// TIA Portal V15.1 export
// export: Created 2024-06-21T08:41:15.862513Z, ExportSetting WithDefaults, DisplayName Totally Integrated Automation Portal, DisplayVersion V15.1 Update 5, DisplayName TIA Portal Openness, DisplayVersion V15.1 Update 5, DisplayName SINAMICS Startdrive Advanced, DisplayVersion V15.1, DisplayName G130, G150, S120, S150, SINAMICS MV, S210, DisplayVersion V15.1, DisplayName G110M, G120, G120C, G120D, G120P, DisplayVersion V15.1, DisplayName STEP 7 Professional, DisplayVersion V15.1 Update 5, DisplayName STEP 7 Safety, DisplayVersion V15.1, DisplayName WinCC Professional, DisplayVersion V15.1 Update 5, DisplayName SIMATIC Visualization Architect, DisplayVersion V15.1
FUNCTION_BLOCK "LGBHoist2Pos2S-C"   // FB6646, FBD
TITLE = LGBHoist2Pos2S-C
{ S7_Optimized_Access := 'TRUE' }
AUTHOR : VCC
FAMILY : Transpor
VERSION : 0.1
// =============================================================================
// This module is used in applications when a Hoist with 2 Positions and two Speeds controlled
// by contactors is needed.
// =============================================================================
// stored: AutoNumber false, IsIECCheckEnabled false, IsRetainMemResEnabled false, MemoryReserve 100, SetENOAutomatically False, UDAEnableTagReadback false
   VAR_INPUT
      I_OverTravelSet { ExternalAccessible := 'False'; ExternalVisible := 'False'; ExternalWritable := 'False'} : Bool;   // Overtravel Switch Set
      I_StopDetSet { ExternalAccessible := 'False'; ExternalVisible := 'False'; ExternalWritable := 'False'} : Bool;   // Stop Detection Set
      I_LowSpeedDetSet { ExternalAccessible := 'False'; ExternalVisible := 'False'; ExternalWritable := 'False'} : Bool;   // Lowspeed Detection Set
      I_LowSpeedDetSetCtrl { ExternalAccessible := 'False'; ExternalVisible := 'False'; ExternalWritable := 'False'} : Bool;   // Lowspeed Detection Set
      I_LowSpeedDetRes { ExternalAccessible := 'False'; ExternalVisible := 'False'; ExternalWritable := 'False'} : Bool;   // Lowspeed Detector Reset
      I_LowSpeedDetResCtrl { ExternalAccessible := 'False'; ExternalVisible := 'False'; ExternalWritable := 'False'} : Bool;   // Lowspeed Detector Reset
      I_StopDetRes { ExternalAccessible := 'False'; ExternalVisible := 'False'; ExternalWritable := 'False'} : Bool;   // Stop Detection Reset
      I_OverTravelRes { ExternalAccessible := 'False'; ExternalVisible := 'False'; ExternalWritable := 'False'} : Bool;   // Overtravel Switch Reset
      I_BypassOvertravelSet { ExternalAccessible := 'False'; ExternalVisible := 'False'; ExternalWritable := 'False'} : Bool;   // Bypass overtravel Set
      I_BypassOvertravelReset { ExternalAccessible := 'False'; ExternalVisible := 'False'; ExternalWritable := 'False'} : Bool;   // Bypass overtravel Reset
      I_BrakeReleased { ExternalAccessible := 'False'; ExternalVisible := 'False'; ExternalWritable := 'False'} : Bool;   // Feedback from brake contactor
      I_SetBegin { ExternalAccessible := 'False'; ExternalVisible := 'False'; ExternalWritable := 'False'} : Bool;   // Condition to start movement Set
      I_ResBegin { ExternalAccessible := 'False'; ExternalVisible := 'False'; ExternalWritable := 'False'} : Bool;   // Condition to start movement Reset
      I_InterlockSetOk { ExternalAccessible := 'False'; ExternalVisible := 'False'; ExternalWritable := 'False'} : Bool;   // Interlock Set Ok
      I_InterlockResetOk { ExternalAccessible := 'False'; ExternalVisible := 'False'; ExternalWritable := 'False'} : Bool;   // Interlock Reset Ok
      I_MotorProtection { ExternalAccessible := 'False'; ExternalVisible := 'False'; ExternalWritable := 'False'} : Bool;   // Motor protection
      I_SafetySwitch { ExternalAccessible := 'False'; ExternalVisible := 'False'; ExternalWritable := 'False'} : Bool;   // Safety Switch
      I_PBSet { ExternalAccessible := 'False'; ExternalVisible := 'False'; ExternalWritable := 'False'} : Bool;   // Push button for manual movememt (on local panel) Set
      I_PBReset { ExternalAccessible := 'False'; ExternalVisible := 'False'; ExternalWritable := 'False'} : Bool;   // Push button for manual movememt (on local panel) Reset
      I_SafetyOk { ExternalAccessible := 'False'; ExternalVisible := 'False'; ExternalWritable := 'False'} : Bool;   // Safety Ok
      I_MotionStopOk { ExternalAccessible := 'False'; ExternalVisible := 'False'; ExternalWritable := 'False'} : Bool;   // Safety Ok / The motion stop is Ok
   END_VAR
   VAR_OUTPUT
      O_SetContactor { ExternalAccessible := 'False'; ExternalVisible := 'False'; ExternalWritable := 'False'} : Bool;   // Activate set contactor / Activate Set Contactor
      O_ResetContactor { ExternalAccessible := 'False'; ExternalVisible := 'False'; ExternalWritable := 'False'} : Bool;   // Activate Reset contactor / Activate Reset Contactor
      O_HSpdContactor { ExternalAccessible := 'False'; ExternalVisible := 'False'; ExternalWritable := 'False'} : Bool;   // Activate High Speed contactor / Activate High Speed Contactor
      O_LSpdContactor { ExternalAccessible := 'False'; ExternalVisible := 'False'; ExternalWritable := 'False'} : Bool;   // Activate low speed contactor / Activate Low Speed Contactor
      O_ReleaseBrake { ExternalAccessible := 'False'; ExternalVisible := 'False'; ExternalWritable := 'False'} : Bool;   // Release the brake of the Motor
      O_ContBypassOvertravelSet { ExternalAccessible := 'False'; ExternalVisible := 'False'; ExternalWritable := 'False'} : Bool;   // Contactor Bypass overtravel Set
      O_ContBypassOvertravelRes { ExternalAccessible := 'False'; ExternalVisible := 'False'; ExternalWritable := 'False'} : Bool;   // Contactor Bypass overtravel Reset
      O_Active { ExternalAccessible := 'False'; ExternalVisible := 'False'; ExternalWritable := 'False'} : Bool;   // Hoist is active
      O_SetFinished { ExternalAccessible := 'False'; ExternalVisible := 'False'; ExternalWritable := 'False'} : Bool;   // Set Position finished
      O_ResFinished { ExternalAccessible := 'False'; ExternalVisible := 'False'; ExternalWritable := 'False'} : Bool;   // Reset Position finished
      O_InSetPos { ExternalAccessible := 'False'; ExternalVisible := 'False'; ExternalWritable := 'False'} : Bool;   // In set Position
      O_InResPos { ExternalAccessible := 'False'; ExternalVisible := 'False'; ExternalWritable := 'False'} : Bool;   // In Reset Position
      O_LEDSet { ExternalAccessible := 'False'; ExternalVisible := 'False'; ExternalWritable := 'False'} : Bool;   // Ledindication / Led indication for Set
      O_LEDRes { ExternalAccessible := 'False'; ExternalVisible := 'False'; ExternalWritable := 'False'} : Bool;   // Ledindication / Led indication for Reset
      O_AlarmABCondition { ExternalAccessible := 'False'; ExternalVisible := 'False'; ExternalWritable := 'False'} : Bool;   // Alarm AB Condition
      O_AlarmA { ExternalAccessible := 'False'; ExternalVisible := 'False'; ExternalWritable := 'False'} : Bool;   // Summation Alarm A
      O_AlarmB { ExternalAccessible := 'False'; ExternalVisible := 'False'; ExternalWritable := 'False'} : Bool;   // Summation Alarm B
      O_AlarmC { ExternalAccessible := 'False'; ExternalVisible := 'False'; ExternalWritable := 'False'} : Bool;   // Summation Alarm C
      O_AlarmD { ExternalAccessible := 'False'; ExternalVisible := 'False'; ExternalWritable := 'False'} : Bool;   // Summation Alarm D
      O_ActualSpeed { ExternalAccessible := 'False'; ExternalVisible := 'False'; ExternalWritable := 'False'} : Real;   // Actual speed value motor
      H_AlarmDWord { ExternalAccessible := 'False'; ExternalVisible := 'False'; ExternalWritable := 'False'} : DWord;   // HMI Alarm Word
   END_VAR
   VAR_IN_OUT
      C_TimeCheckSpeedOK { ExternalAccessible := 'False'; ExternalVisible := 'False'; ExternalWritable := 'False'} : DInt := 2000;   // Time check speed OK
      IO_Modes : "Modes";   // Modes
      H_HMI : "H_HMI";   // Animation
      "H_GBHoist2Pos2S-C" : "H_GBHoist2Pos2S-C";   // Animation
      C_Config : "Hoist2Pos2S-C-Config";   // Config
   END_VAR
   VAR
      _Motor { ExternalAccessible := 'False'; ExternalVisible := 'False'; ExternalWritable := 'False'} : "LGBMotor2W2S-C";
      H_FncSelInHMI { ExternalAccessible := 'False'; ExternalVisible := 'False'; ExternalWritable := 'False'} : Bool;
      AlarmABCondition { ExternalAccessible := 'False'; ExternalVisible := 'False'; ExternalWritable := 'False'} : Bool;   // Alarm AB Condition
      AA_MotorProtection { ExternalAccessible := 'False'; ExternalVisible := 'False'; ExternalWritable := 'False'} : Bool;   // Motorprotection Tripped
      AA_SafetySwitch { ExternalAccessible := 'False'; ExternalVisible := 'False'; ExternalWritable := 'False'} : Bool;   // Safety Switch Not Ok
      AB_OverTravelSet { ExternalAccessible := 'False'; ExternalVisible := 'False'; ExternalWritable := 'False'} : Bool;   // Overtravel Set
      AB_OverTravelRes { ExternalAccessible := 'False'; ExternalVisible := 'False'; ExternalWritable := 'False'} : Bool;   // Overtravel Reset
      AB_LSpDetSet { ExternalAccessible := 'False'; ExternalVisible := 'False'; ExternalWritable := 'False'} : Bool;   // Low Speed Detector Set Missing
      AB_LSpDetSetCtrl { ExternalAccessible := 'False'; ExternalVisible := 'False'; ExternalWritable := 'False'} : Bool;   // Low Speed Detector Ctrl Set Missing
      AB_LSpDetRes { ExternalAccessible := 'False'; ExternalVisible := 'False'; ExternalWritable := 'False'} : Bool;   // Low Speed Detector Reset Missing
      AB_LSpDetResCtrl { ExternalAccessible := 'False'; ExternalVisible := 'False'; ExternalWritable := 'False'} : Bool;   // Low Speed Detector Ctrl Reset Missing
      AB_BrakeFbk { ExternalAccessible := 'False'; ExternalVisible := 'False'; ExternalWritable := 'False'} : Bool;   // Safety Switch Not Ok / Brake feedback Nok / Säkerhetsbrytare Ej Ok
      AC_OvtSetAlm { ExternalAccessible := 'False'; ExternalVisible := 'False'; ExternalWritable := 'False'} : Bool;   // Timeout Set
      AC_OvtResAlm { ExternalAccessible := 'False'; ExternalVisible := 'False'; ExternalWritable := 'False'} : Bool;   // Timeout Reset
      AC_OvertravelSetBypassAlm { ExternalAccessible := 'False'; ExternalVisible := 'False'; ExternalWritable := 'False'} : Bool;   // Overtravel Set Bypass
      AC_OvertravelResBypassAlm { ExternalAccessible := 'False'; ExternalVisible := 'False'; ExternalWritable := 'False'} : Bool;   // Overtravel Reset Bypass
      AD_IntlkSet { ExternalAccessible := 'False'; ExternalVisible := 'False'; ExternalWritable := 'False'} : Bool;   // Interlock Not Ok
      AD_IntlkRes { ExternalAccessible := 'False'; ExternalVisible := 'False'; ExternalWritable := 'False'} : Bool;   // Interlock Not Ok
      AC_LiftNoPos { ExternalAccessible := 'False'; ExternalVisible := 'False'; ExternalWritable := 'False'} : Bool;   // Lifter Not in position
      AD_MotionStop { ExternalAccessible := 'False'; ExternalVisible := 'False'; ExternalWritable := 'False'} : Bool;   // Motion Stop
      SafetyOk { ExternalAccessible := 'False'; ExternalVisible := 'False'; ExternalWritable := 'False'} : Bool;   // Safety Ok
      AlarmA { ExternalAccessible := 'False'; ExternalVisible := 'False'; ExternalWritable := 'False'} : Bool;   // Alarm A
      AlarmB { ExternalAccessible := 'False'; ExternalVisible := 'False'; ExternalWritable := 'False'} : Bool;   // Alarm B
      AlarmC { ExternalAccessible := 'False'; ExternalVisible := 'False'; ExternalWritable := 'False'} : Bool;   // Alarm C
      AlarmD { ExternalAccessible := 'False'; ExternalVisible := 'False'; ExternalWritable := 'False'} : Bool;   // Alarm D
      LSpdContactor { ExternalAccessible := 'False'; ExternalVisible := 'False'; ExternalWritable := 'False'} : Bool;   // Contactor low speed / Activate Low Speed Contactor
      HSpdContactor { ExternalAccessible := 'False'; ExternalVisible := 'False'; ExternalWritable := 'False'} : Bool;   // Contactor High Speed / Activate High Speed Contactor
      SetContactor { ExternalAccessible := 'False'; ExternalVisible := 'False'; ExternalWritable := 'False'} : Bool;   // Activate Set Contactor
      ResetContactor { ExternalAccessible := 'False'; ExternalVisible := 'False'; ExternalWritable := 'False'} : Bool;   // Activate Reset Contactor
      ReleaseBrake { ExternalAccessible := 'False'; ExternalVisible := 'False'; ExternalWritable := 'False'} : Bool;   // Activate Reset contactor / Release Brake
      MotorLoopActive { ExternalAccessible := 'False'; ExternalVisible := 'False'; ExternalWritable := 'False'} : Bool;   // Motor Loop Active
      MotorCmdLSpdSet { ExternalAccessible := 'False'; ExternalVisible := 'False'; ExternalWritable := 'False'} : Bool;   // Command to Motorloop low Speed Set
      MotorCmdLSpdRes { ExternalAccessible := 'False'; ExternalVisible := 'False'; ExternalWritable := 'False'} : Bool;   // Command to Motorloop low speed Reset
      MotorCmdHSpdSet { ExternalAccessible := 'False'; ExternalVisible := 'False'; ExternalWritable := 'False'} : Bool;   // Command to Motorloop high Speed Set
      MotorCmdHSpdRes { ExternalAccessible := 'False'; ExternalVisible := 'False'; ExternalWritable := 'False'} : Bool;   // Command to Motorloop high speed Reset
      MotorReqLSpdSet { ExternalAccessible := 'False'; ExternalVisible := 'False'; ExternalWritable := 'False'} : Bool;   // Request low Speed Set
      MotorReqLSpdRes { ExternalAccessible := 'False'; ExternalVisible := 'False'; ExternalWritable := 'False'} : Bool;   // Request low speed Reset
      MotorReqHSpdSet { ExternalAccessible := 'False'; ExternalVisible := 'False'; ExternalWritable := 'False'} : Bool;   // Request highSpeed Set
      MotorReqHSpdRes { ExternalAccessible := 'False'; ExternalVisible := 'False'; ExternalWritable := 'False'} : Bool;   // Request high speed Reset
      ManHighSpdSel { ExternalAccessible := 'False'; ExternalVisible := 'False'; ExternalWritable := 'False'} : Bool;   // Low speed selected in manual
      HSpdMem { ExternalAccessible := 'False'; ExternalVisible := 'False'; ExternalWritable := 'False'} : Bool;   // High speed memory flag
      BlockHSpeed { ExternalAccessible := 'False'; ExternalVisible := 'False'; ExternalWritable := 'False'} : Bool;   // AND of ALL detections
      AlarmABAct { ExternalAccessible := 'False'; ExternalVisible := 'False'; ExternalWritable := 'False'} : Bool;   // Alarm A or B is active
      OverTravelSetAlmCond { ExternalAccessible := 'False'; ExternalVisible := 'False'; ExternalWritable := 'False'} : Bool;   // Alarm AB Condition
      OverTravelResAlmCond { ExternalAccessible := 'False'; ExternalVisible := 'False'; ExternalWritable := 'False'} : Bool;   // Alarm AB Condition
      MotorLoopAlmCond { ExternalAccessible := 'False'; ExternalVisible := 'False'; ExternalWritable := 'False'} : Bool;   // Alarm AB Condition
      CmdSet { ExternalAccessible := 'False'; ExternalVisible := 'False'; ExternalWritable := 'False'} : Bool;   // Activate Set (up) command
      CmdRes { ExternalAccessible := 'False'; ExternalVisible := 'False'; ExternalWritable := 'False'} : Bool;   // Activate Reset (down) command
      InSetPos { ExternalAccessible := 'False'; ExternalVisible := 'False'; ExternalWritable := 'False'} : Bool;   // In set Position
      InResPos { ExternalAccessible := 'False'; ExternalVisible := 'False'; ExternalWritable := 'False'} : Bool;   // In Reset Position
      TimeOutNotDownCmd { ExternalAccessible := 'False'; ExternalVisible := 'False'; ExternalWritable := 'False'} : Bool;   // Timer result
      TimeOutNotUpCmd { ExternalAccessible := 'False'; ExternalVisible := 'False'; ExternalWritable := 'False'} : Bool;   // Timer result
      _TimerNoDownCmd { ExternalAccessible := 'False'; ExternalVisible := 'False'; ExternalWritable := 'False'} : "LTimer";   // FB
      _TimerNoUpCmd { ExternalAccessible := 'False'; ExternalVisible := 'False'; ExternalWritable := 'False'} : "LTimer";   // FB
      _TimerNoPos { ExternalAccessible := 'False'; ExternalVisible := 'False'; ExternalWritable := 'False'} : "LTimer";
      _BypassOvertravelSet { ExternalAccessible := 'False'; ExternalVisible := 'False'; ExternalWritable := 'False'} : "L1AlarmMultiIn";   // FB
      _BypassOvertravelReset { ExternalAccessible := 'False'; ExternalVisible := 'False'; ExternalWritable := 'False'} : "L1AlarmMultiIn";   // FB
      _OverTravelSet { ExternalAccessible := 'False'; ExternalVisible := 'False'; ExternalWritable := 'False'} : "L1AlarmMultiIn";
      _OverTravelRes { ExternalAccessible := 'False'; ExternalVisible := 'False'; ExternalWritable := 'False'} : "L1AlarmMultiIn";
      _OvtSetAlmTimer { ExternalAccessible := 'False'; ExternalVisible := 'False'; ExternalWritable := 'False'} : "LTimer";   // FB
      _OvtResAlmTimer { ExternalAccessible := 'False'; ExternalVisible := 'False'; ExternalWritable := 'False'} : "LTimer";   // FB
      Edge { ExternalAccessible := 'False'; ExternalVisible := 'False'; ExternalWritable := 'False'} : Array[1..8] of Bool;   // Edge
   END_VAR
   VAR_TEMP
      NotUsedH_HMI : "H_HMI";   // Temp
      H_HMIMotor : "H_HMI";   // Temp
      HMICMD : "ConvHMICMD";   // Temp
   END_VAR
   VAR_TEMP   // added for the SCL form of the ladder/FBD networks
      _w1 : Bool;
   END_VAR
BEGIN

REGION Network 1: **** 1 - Inputs **** HMI Commands
   // HMI Commands
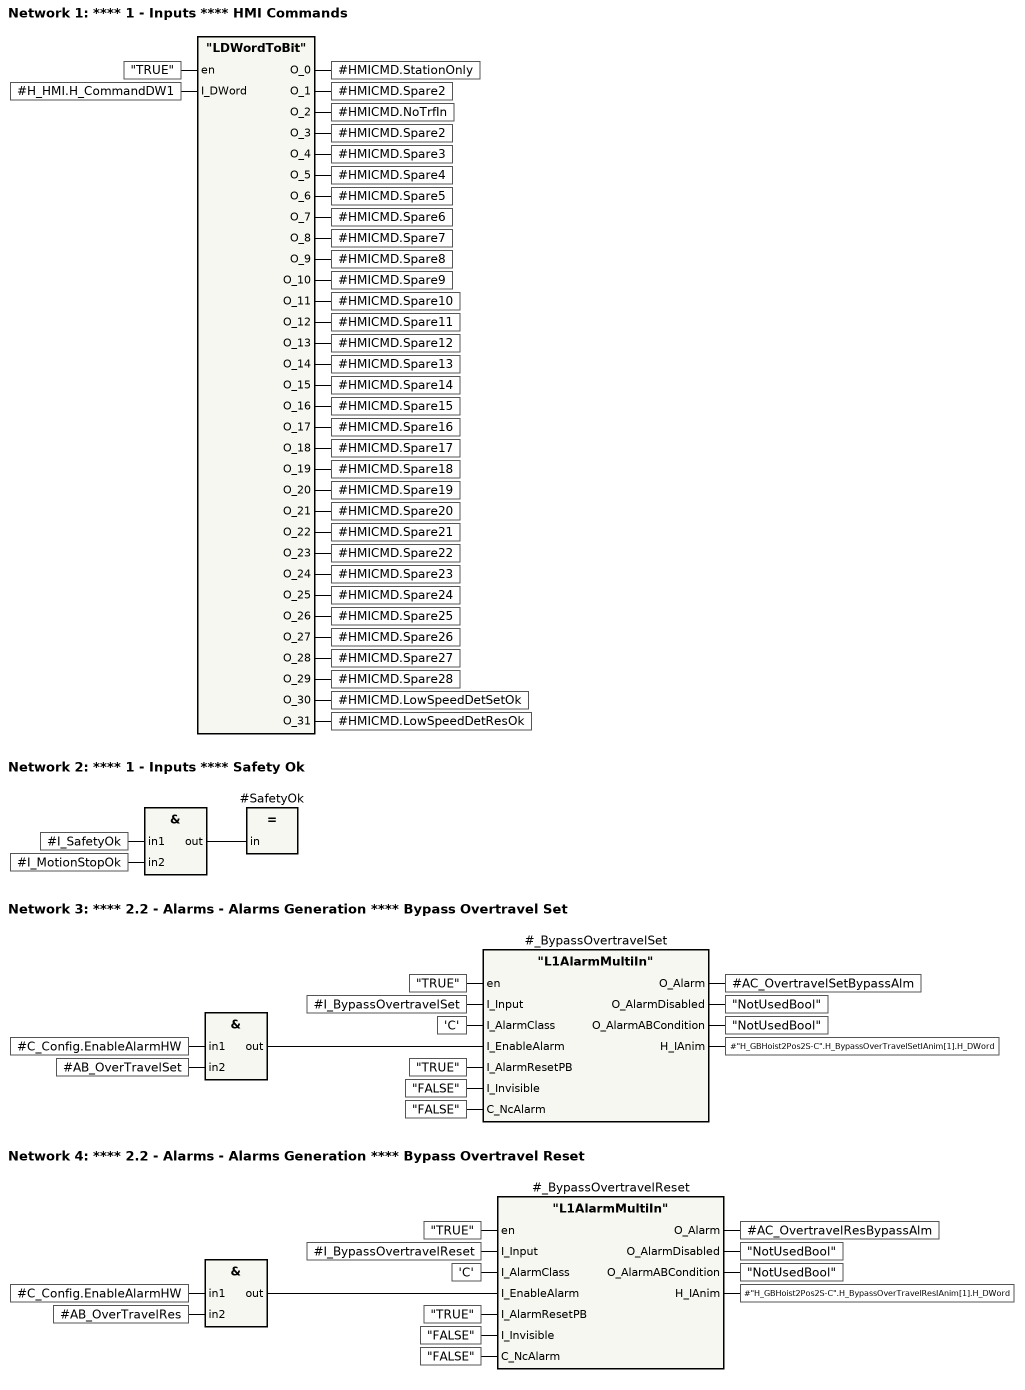
   IF "TRUE" THEN
       "LDWordToBit"(I_DWord := #H_HMI.H_CommandDW1,
                     O_0 => #HMICMD.StationOnly,
                     O_1 => #HMICMD.Spare2,
                     O_2 => #HMICMD.NoTrfIn,
                     O_3 => #HMICMD.Spare2,
                     O_4 => #HMICMD.Spare3,
                     O_5 => #HMICMD.Spare4,
                     O_6 => #HMICMD.Spare5,
                     O_7 => #HMICMD.Spare6,
                     O_8 => #HMICMD.Spare7,
                     O_9 => #HMICMD.Spare8,
                     O_10 => #HMICMD.Spare9,
                     O_11 => #HMICMD.Spare10,
                     O_12 => #HMICMD.Spare11,
                     O_13 => #HMICMD.Spare12,
                     O_14 => #HMICMD.Spare13,
                     O_15 => #HMICMD.Spare14,
                     O_16 => #HMICMD.Spare15,
                     O_17 => #HMICMD.Spare16,
                     O_18 => #HMICMD.Spare17,
                     O_19 => #HMICMD.Spare18,
                     O_20 => #HMICMD.Spare19,
                     O_21 => #HMICMD.Spare20,
                     O_22 => #HMICMD.Spare21,
                     O_23 => #HMICMD.Spare22,
                     O_24 => #HMICMD.Spare23,
                     O_25 => #HMICMD.Spare24,
                     O_26 => #HMICMD.Spare25,
                     O_27 => #HMICMD.Spare26,
                     O_28 => #HMICMD.Spare27,
                     O_29 => #HMICMD.Spare28,
                     O_30 => #HMICMD.LowSpeedDetSetOk,
                     O_31 => #HMICMD.LowSpeedDetResOk);
   END_IF;
END_REGION

REGION Network 2: **** 1 - Inputs **** Safety Ok
   #SafetyOk := #I_SafetyOk AND #I_MotionStopOk;
END_REGION

REGION Network 3: **** 2.2 - Alarms - Alarms Generation **** Bypass Overtravel Set
   // Alarm Bypass Overtravel Set
   IF "TRUE" THEN
       #_BypassOvertravelSet(I_Input := #I_BypassOvertravelSet,   // "L1AlarmMultiIn"
                             I_AlarmClass := 'C',
                             I_EnableAlarm := #C_Config.EnableAlarmHW AND #AB_OverTravelSet,
                             I_AlarmResetPB := "TRUE",
                             I_Invisible := "FALSE",
                             C_NcAlarm := "FALSE",
                             O_Alarm => #AC_OvertravelSetBypassAlm,
                             O_AlarmDisabled => "NotUsedBool",
                             O_AlarmABCondition => "NotUsedBool",
                             H_IAnim => #"H_GBHoist2Pos2S-C".H_BypassOverTravelSetIAnim[1].H_DWord);
   END_IF;
END_REGION

REGION Network 4: **** 2.2 - Alarms - Alarms Generation **** Bypass Overtravel Reset
   // Alarm Bypass Overtravel Reset
   IF "TRUE" THEN
       #_BypassOvertravelReset(I_Input := #I_BypassOvertravelReset,   // "L1AlarmMultiIn"
                               I_AlarmClass := 'C',
                               I_EnableAlarm := #C_Config.EnableAlarmHW AND #AB_OverTravelRes,
                               I_AlarmResetPB := "TRUE",
                               I_Invisible := "FALSE",
                               C_NcAlarm := "FALSE",
                               O_Alarm => #AC_OvertravelResBypassAlm,
                               O_AlarmDisabled => "NotUsedBool",
                               O_AlarmABCondition => "NotUsedBool",
                               H_IAnim => #"H_GBHoist2Pos2S-C".H_BypassOverTravelResIAnim[1].H_DWord);
   END_IF;
END_REGION

REGION Network 5: **** 2.2 - Alarms - Alarms Generation **** Over Travel Set Alarm
   // Over Travel Set Alarm
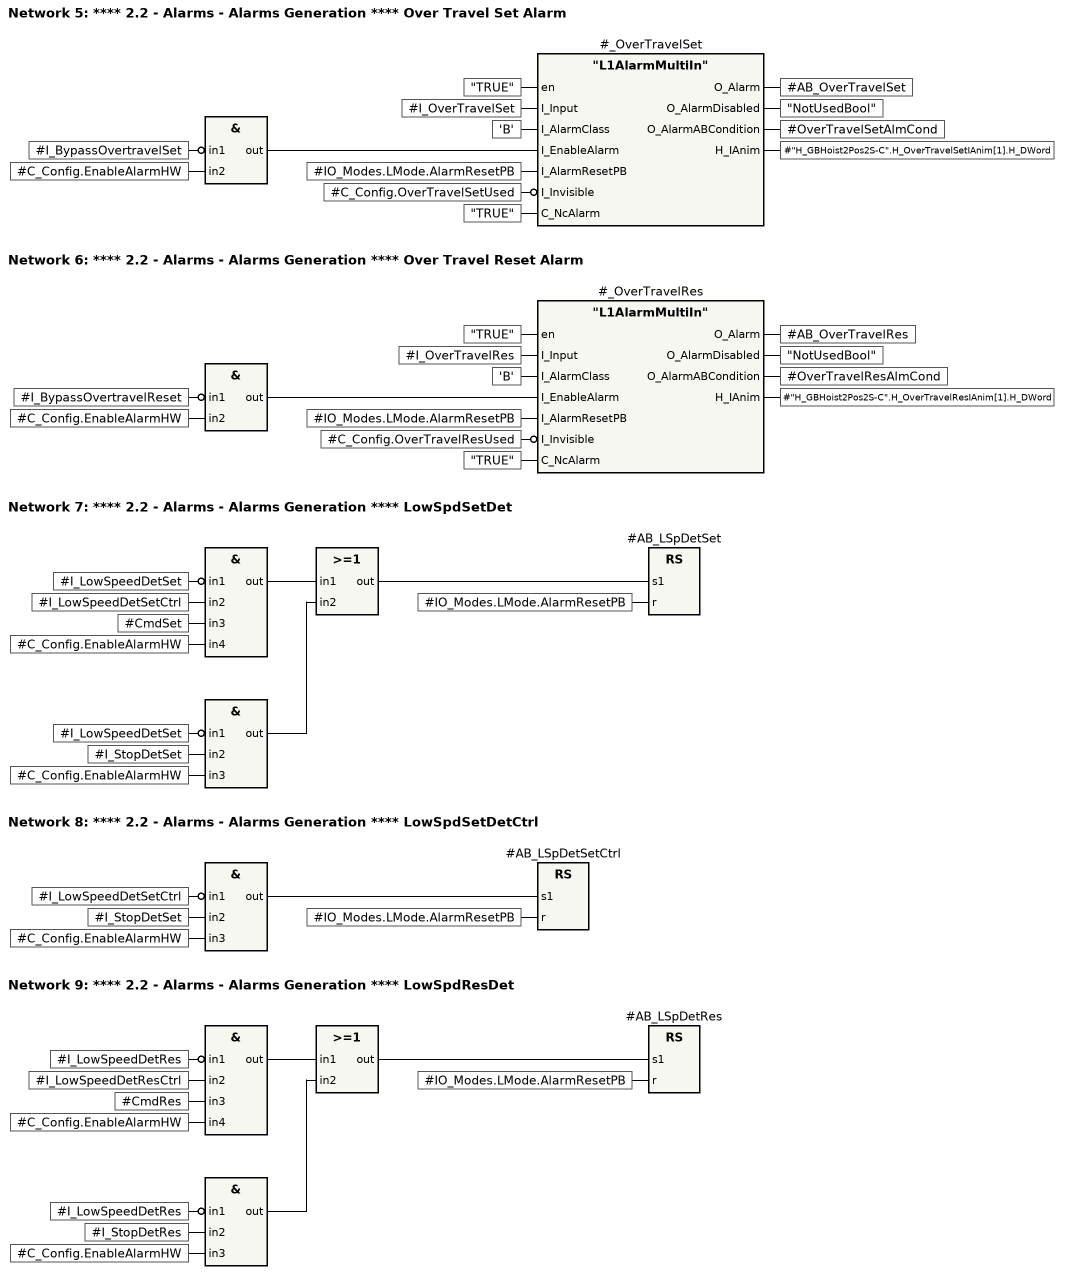
   IF "TRUE" THEN
       #_OverTravelSet(I_Input := #I_OverTravelSet,   // "L1AlarmMultiIn"
                       I_AlarmClass := 'B',
                       I_EnableAlarm := NOT #I_BypassOvertravelSet AND #C_Config.EnableAlarmHW,
                       I_AlarmResetPB := #IO_Modes.LMode.AlarmResetPB,
                       I_Invisible := NOT #C_Config.OverTravelSetUsed,
                       C_NcAlarm := "TRUE",
                       O_Alarm => #AB_OverTravelSet,
                       O_AlarmDisabled => "NotUsedBool",
                       O_AlarmABCondition => #OverTravelSetAlmCond,
                       H_IAnim => #"H_GBHoist2Pos2S-C".H_OverTravelSetIAnim[1].H_DWord);
   END_IF;
END_REGION

REGION Network 6: **** 2.2 - Alarms - Alarms Generation **** Over Travel Reset Alarm
   // Over Travel Reset Alarm
   IF "TRUE" THEN
       #_OverTravelRes(I_Input := #I_OverTravelRes,   // "L1AlarmMultiIn"
                       I_AlarmClass := 'B',
                       I_EnableAlarm := NOT #I_BypassOvertravelReset AND #C_Config.EnableAlarmHW,
                       I_AlarmResetPB := #IO_Modes.LMode.AlarmResetPB,
                       I_Invisible := NOT #C_Config.OverTravelResUsed,
                       C_NcAlarm := "TRUE",
                       O_Alarm => #AB_OverTravelRes,
                       O_AlarmDisabled => "NotUsedBool",
                       O_AlarmABCondition => #OverTravelResAlmCond,
                       H_IAnim => #"H_GBHoist2Pos2S-C".H_OverTravelResIAnim[1].H_DWord);
   END_IF;
END_REGION

REGION Network 7: **** 2.2 - Alarms - Alarms Generation **** LowSpdSetDet
   // Alarm Lift low Speed Set  detector
   IF #IO_Modes.LMode.AlarmResetPB THEN
       #AB_LSpDetSet := FALSE;   // RS flip-flop
   END_IF;
   IF (NOT #I_LowSpeedDetSet AND #I_LowSpeedDetSetCtrl AND #CmdSet AND #C_Config.EnableAlarmHW) OR (NOT #I_LowSpeedDetSet AND #I_StopDetSet AND #C_Config.EnableAlarmHW) THEN
       #AB_LSpDetSet := TRUE;
   END_IF;
END_REGION

REGION Network 8: **** 2.2 - Alarms - Alarms Generation **** LowSpdSetDetCtrl
   // Alarm Lift low Speed Set Ctrl detector
   IF #IO_Modes.LMode.AlarmResetPB THEN
       #AB_LSpDetSetCtrl := FALSE;   // RS flip-flop
   END_IF;
   IF NOT #I_LowSpeedDetSetCtrl AND #I_StopDetSet AND #C_Config.EnableAlarmHW THEN
       #AB_LSpDetSetCtrl := TRUE;
   END_IF;
END_REGION

REGION Network 9: **** 2.2 - Alarms - Alarms Generation **** LowSpdResDet
   // Alarm Lift low speed Reset  detector
   IF #IO_Modes.LMode.AlarmResetPB THEN
       #AB_LSpDetRes := FALSE;   // RS flip-flop
   END_IF;
   IF (NOT #I_LowSpeedDetRes AND #I_LowSpeedDetResCtrl AND #CmdRes AND #C_Config.EnableAlarmHW) OR (NOT #I_LowSpeedDetRes AND #I_StopDetRes AND #C_Config.EnableAlarmHW) THEN
       #AB_LSpDetRes := TRUE;
   END_IF;
END_REGION

REGION Network 10: **** 2.2 - Alarms - Alarms Generation **** LowSpdResDet Ctrl
   // Alarm Lift low speed Reset Ctrl detector
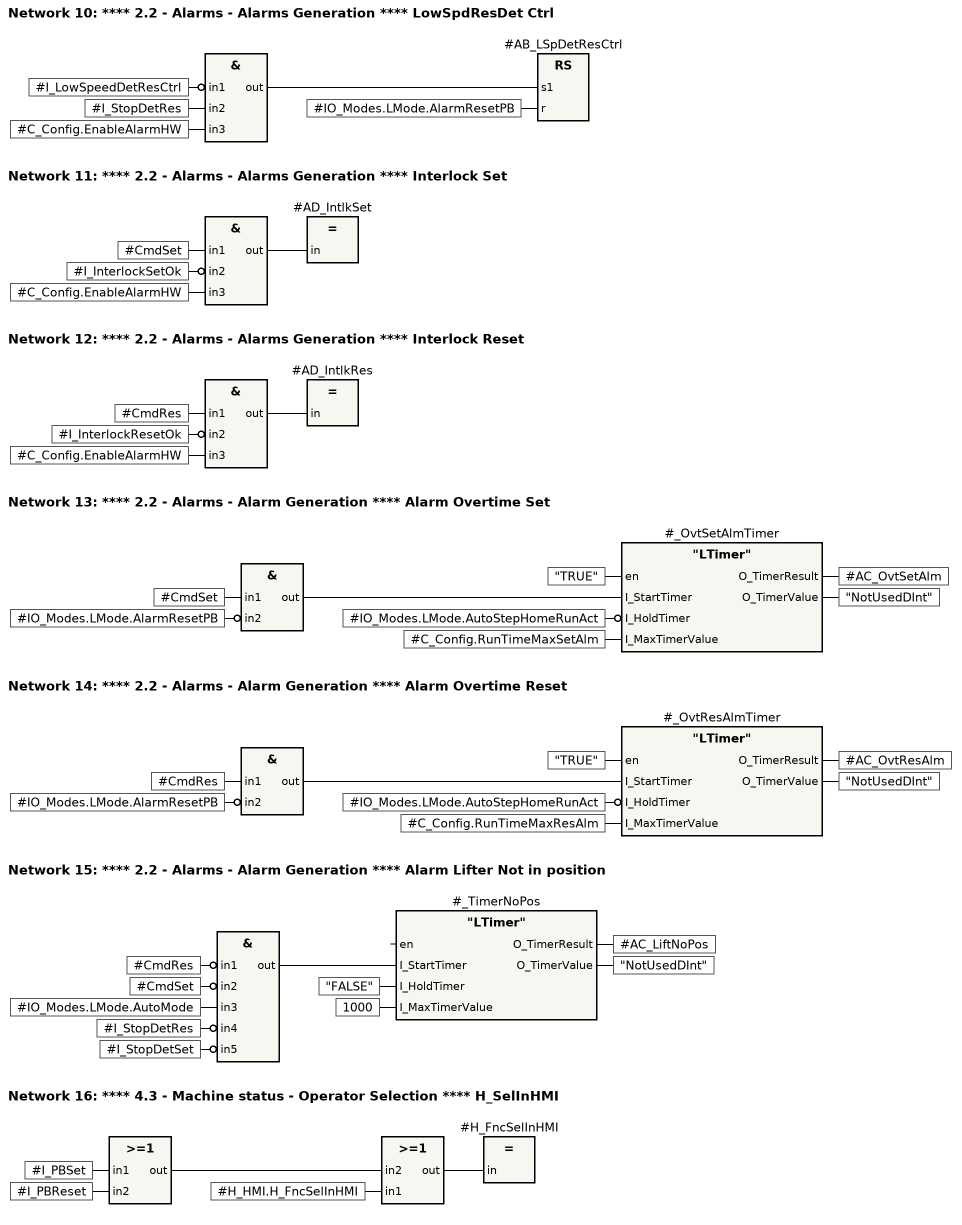
   IF #IO_Modes.LMode.AlarmResetPB THEN
       #AB_LSpDetResCtrl := FALSE;   // RS flip-flop
   END_IF;
   IF NOT #I_LowSpeedDetResCtrl AND #I_StopDetRes AND #C_Config.EnableAlarmHW THEN
       #AB_LSpDetResCtrl := TRUE;
   END_IF;
END_REGION

REGION Network 11: **** 2.2 - Alarms - Alarms Generation **** Interlock Set
   // Alarm Interlock Set
   #AD_IntlkSet := #CmdSet AND NOT #I_InterlockSetOk AND #C_Config.EnableAlarmHW;
END_REGION

REGION Network 12: **** 2.2 - Alarms - Alarms Generation **** Interlock Reset
   // Alarm Interlock Reset
   #AD_IntlkRes := #CmdRes AND NOT #I_InterlockResetOk AND #C_Config.EnableAlarmHW;
END_REGION

REGION Network 13: **** 2.2 - Alarms - Alarm Generation **** Alarm Overtime Set
   // Alarm Overtime Set
   IF "TRUE" THEN
       #_OvtSetAlmTimer(I_StartTimer := #CmdSet AND NOT #IO_Modes.LMode.AlarmResetPB,   // "LTimer"
                        I_HoldTimer := NOT #IO_Modes.LMode.AutoStepHomeRunAct,
                        I_MaxTimerValue := #C_Config.RunTimeMaxSetAlm,
                        O_TimerResult => #AC_OvtSetAlm,
                        O_TimerValue => "NotUsedDInt");
   END_IF;
END_REGION

REGION Network 14: **** 2.2 - Alarms - Alarm Generation **** Alarm Overtime Reset
   // Alarm Overtime Set
   IF "TRUE" THEN
       #_OvtResAlmTimer(I_StartTimer := #CmdRes AND NOT #IO_Modes.LMode.AlarmResetPB,   // "LTimer"
                        I_HoldTimer := NOT #IO_Modes.LMode.AutoStepHomeRunAct,
                        I_MaxTimerValue := #C_Config.RunTimeMaxResAlm,
                        O_TimerResult => #AC_OvtResAlm,
                        O_TimerValue => "NotUsedDInt");
   END_IF;
END_REGION

REGION Network 15: **** 2.2 - Alarms - Alarm Generation **** Alarm Lifter Not in position
   // Alarm Lifter Not in position
   #_TimerNoPos(I_StartTimer := NOT #CmdRes AND NOT #CmdSet AND #IO_Modes.LMode.AutoMode AND NOT #I_StopDetRes AND NOT #I_StopDetSet,   // "LTimer"
                I_HoldTimer := "FALSE",
                I_MaxTimerValue := 1000,
                O_TimerResult => #AC_LiftNoPos,
                O_TimerValue => "NotUsedDInt");
END_REGION

REGION Network 16: **** 4.3 - Machine status - Operator Selection **** H_SelInHMI
   #H_FncSelInHMI := #I_PBSet OR #I_PBReset OR #H_HMI.H_FncSelInHMI;
END_REGION

REGION Network 17: **** 4.3 - Machine status - Operator Selection **** Reset H_SelInHMI
   // Reset H_SelInHMI
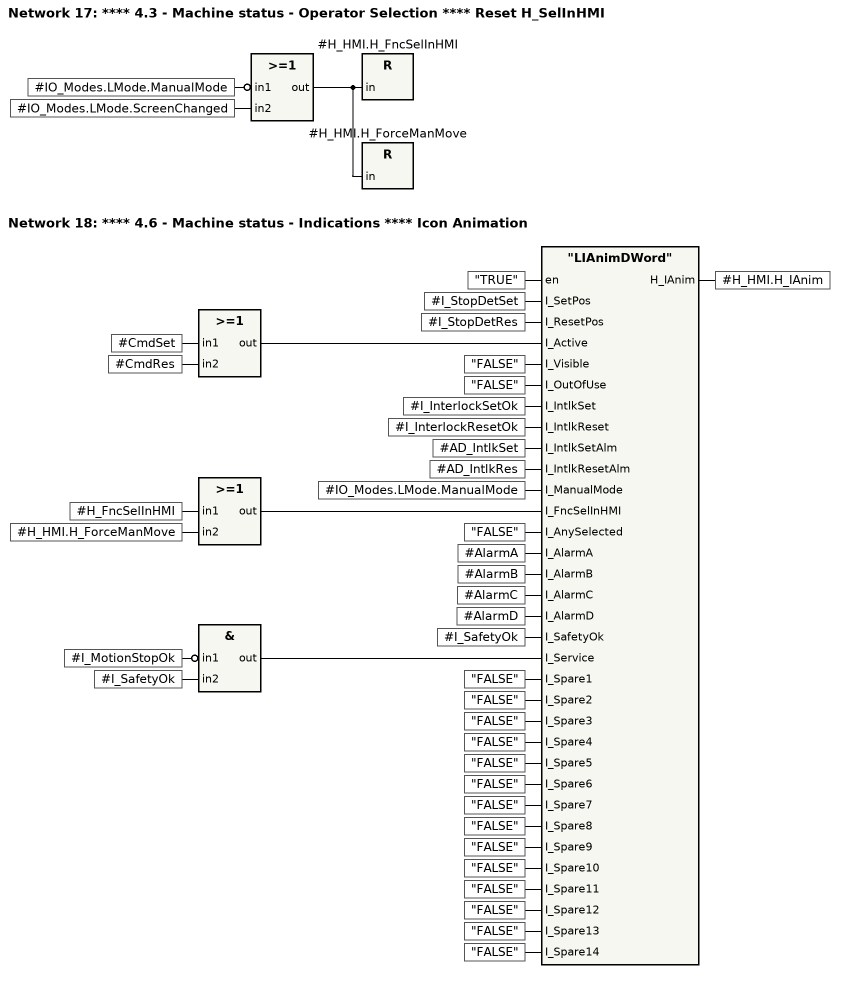
   IF NOT #IO_Modes.LMode.ManualMode OR #IO_Modes.LMode.ScreenChanged THEN
       #H_HMI.H_FncSelInHMI := FALSE;
       #H_HMI.H_ForceManMove := FALSE;
   END_IF;
END_REGION

REGION Network 18: **** 4.6 - Machine status - Indications **** Icon Animation
   // Animation for HMI
   IF "TRUE" THEN
       "LIAnimDWord"(I_SetPos := #I_StopDetSet,
                     I_ResetPos := #I_StopDetRes,
                     I_Active := #CmdSet OR #CmdRes,
                     I_Visible := "FALSE",
                     I_OutOfUse := "FALSE",
                     I_IntlkSet := #I_InterlockSetOk,
                     I_IntlkReset := #I_InterlockResetOk,
                     I_IntlkSetAlm := #AD_IntlkSet,
                     I_IntlkResetAlm := #AD_IntlkRes,
                     I_ManualMode := #IO_Modes.LMode.ManualMode,
                     I_FncSelInHMI := #H_FncSelInHMI OR #H_HMI.H_ForceManMove,
                     I_AnySelected := "FALSE",
                     I_AlarmA := #AlarmA,
                     I_AlarmB := #AlarmB,
                     I_AlarmC := #AlarmC,
                     I_AlarmD := #AlarmD,
                     I_SafetyOk := #I_SafetyOk,
                     I_Service := NOT #I_MotionStopOk AND #I_SafetyOk,
                     I_Spare1 := "FALSE",
                     I_Spare2 := "FALSE",
                     I_Spare3 := "FALSE",
                     I_Spare4 := "FALSE",
                     I_Spare5 := "FALSE",
                     I_Spare6 := "FALSE",
                     I_Spare7 := "FALSE",
                     I_Spare8 := "FALSE",
                     I_Spare9 := "FALSE",
                     I_Spare10 := "FALSE",
                     I_Spare11 := "FALSE",
                     I_Spare12 := "FALSE",
                     I_Spare13 := "FALSE",
                     I_Spare14 := "FALSE",
                     H_IAnim => #H_HMI.H_IAnim);
   END_IF;
END_REGION

REGION Network 19: **** 4.6 - Machine status - Indications **** StopDetSetIAnim
   // Stop detector set animation
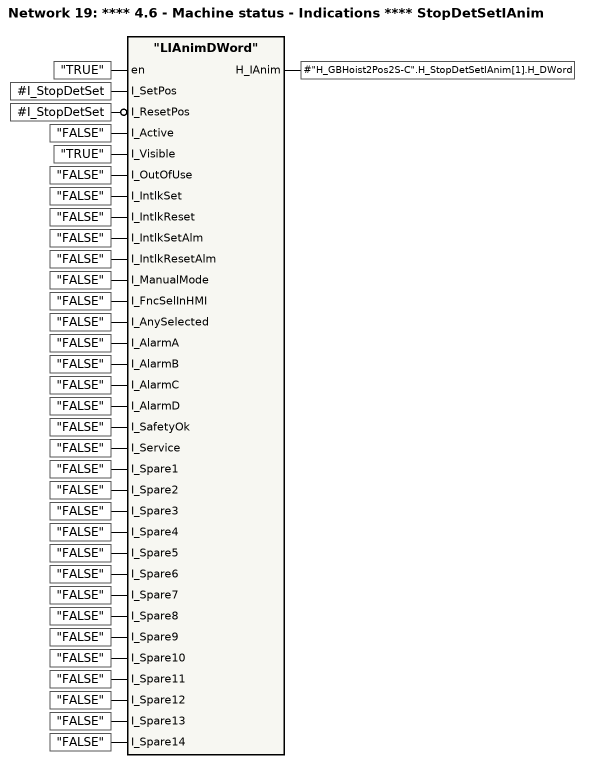
   IF "TRUE" THEN
       "LIAnimDWord"(I_SetPos := #I_StopDetSet,
                     I_ResetPos := NOT #I_StopDetSet,
                     I_Active := "FALSE",
                     I_Visible := "TRUE",
                     I_OutOfUse := "FALSE",
                     I_IntlkSet := "FALSE",
                     I_IntlkReset := "FALSE",
                     I_IntlkSetAlm := "FALSE",
                     I_IntlkResetAlm := "FALSE",
                     I_ManualMode := "FALSE",
                     I_FncSelInHMI := "FALSE",
                     I_AnySelected := "FALSE",
                     I_AlarmA := "FALSE",
                     I_AlarmB := "FALSE",
                     I_AlarmC := "FALSE",
                     I_AlarmD := "FALSE",
                     I_SafetyOk := "FALSE",
                     I_Service := "FALSE",
                     I_Spare1 := "FALSE",
                     I_Spare2 := "FALSE",
                     I_Spare3 := "FALSE",
                     I_Spare4 := "FALSE",
                     I_Spare5 := "FALSE",
                     I_Spare6 := "FALSE",
                     I_Spare7 := "FALSE",
                     I_Spare8 := "FALSE",
                     I_Spare9 := "FALSE",
                     I_Spare10 := "FALSE",
                     I_Spare11 := "FALSE",
                     I_Spare12 := "FALSE",
                     I_Spare13 := "FALSE",
                     I_Spare14 := "FALSE",
                     H_IAnim => #"H_GBHoist2Pos2S-C".H_StopDetSetIAnim[1].H_DWord);
   END_IF;
END_REGION

REGION Network 20: **** 4.6 - Machine status - Indications **** LSpeedDetSetIAnim
   // Low Speed Set detector animation
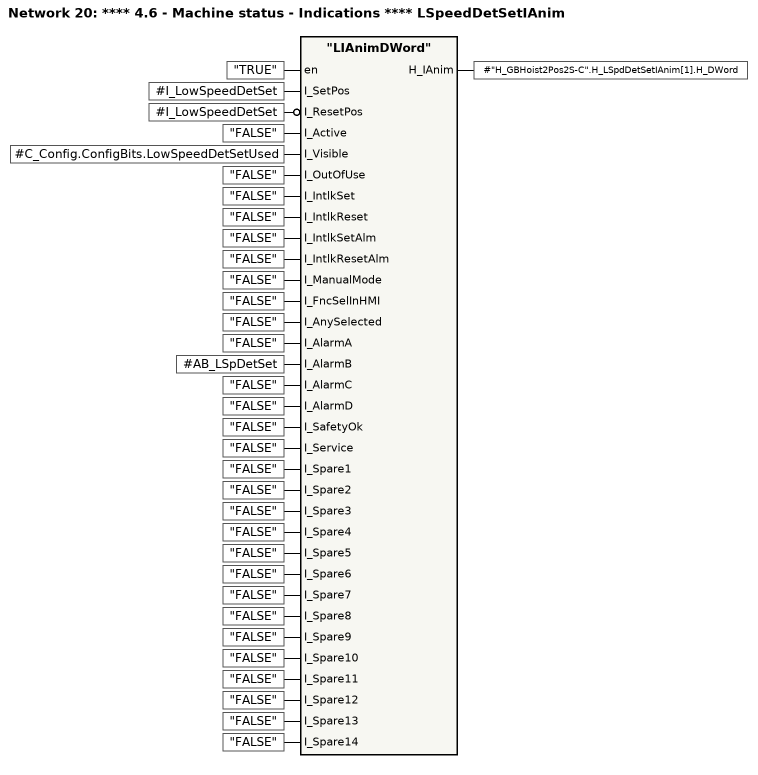
   IF "TRUE" THEN
       "LIAnimDWord"(I_SetPos := #I_LowSpeedDetSet,
                     I_ResetPos := NOT #I_LowSpeedDetSet,
                     I_Active := "FALSE",
                     I_Visible := #C_Config.ConfigBits.LowSpeedDetSetUsed,
                     I_OutOfUse := "FALSE",
                     I_IntlkSet := "FALSE",
                     I_IntlkReset := "FALSE",
                     I_IntlkSetAlm := "FALSE",
                     I_IntlkResetAlm := "FALSE",
                     I_ManualMode := "FALSE",
                     I_FncSelInHMI := "FALSE",
                     I_AnySelected := "FALSE",
                     I_AlarmA := "FALSE",
                     I_AlarmB := #AB_LSpDetSet,
                     I_AlarmC := "FALSE",
                     I_AlarmD := "FALSE",
                     I_SafetyOk := "FALSE",
                     I_Service := "FALSE",
                     I_Spare1 := "FALSE",
                     I_Spare2 := "FALSE",
                     I_Spare3 := "FALSE",
                     I_Spare4 := "FALSE",
                     I_Spare5 := "FALSE",
                     I_Spare6 := "FALSE",
                     I_Spare7 := "FALSE",
                     I_Spare8 := "FALSE",
                     I_Spare9 := "FALSE",
                     I_Spare10 := "FALSE",
                     I_Spare11 := "FALSE",
                     I_Spare12 := "FALSE",
                     I_Spare13 := "FALSE",
                     I_Spare14 := "FALSE",
                     H_IAnim => #"H_GBHoist2Pos2S-C".H_LSpdDetSetIAnim[1].H_DWord);
   END_IF;
END_REGION

REGION Network 21: **** 4.6 - Machine status - Indications **** LSpeedDetSetCtrlIAnim
   // Low speed detector Set Control animation
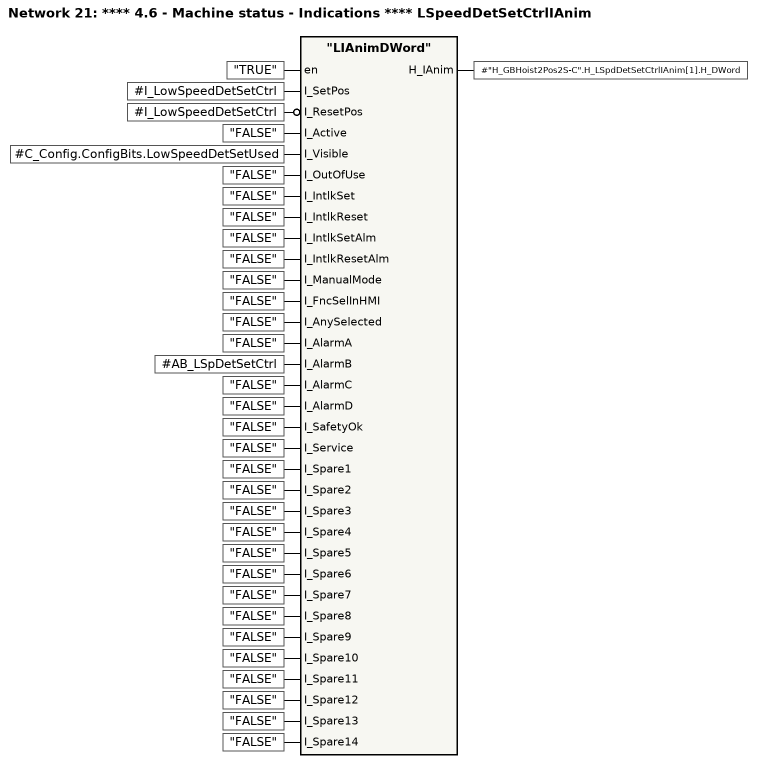
   IF "TRUE" THEN
       "LIAnimDWord"(I_SetPos := #I_LowSpeedDetSetCtrl,
                     I_ResetPos := NOT #I_LowSpeedDetSetCtrl,
                     I_Active := "FALSE",
                     I_Visible := #C_Config.ConfigBits.LowSpeedDetSetUsed,
                     I_OutOfUse := "FALSE",
                     I_IntlkSet := "FALSE",
                     I_IntlkReset := "FALSE",
                     I_IntlkSetAlm := "FALSE",
                     I_IntlkResetAlm := "FALSE",
                     I_ManualMode := "FALSE",
                     I_FncSelInHMI := "FALSE",
                     I_AnySelected := "FALSE",
                     I_AlarmA := "FALSE",
                     I_AlarmB := #AB_LSpDetSetCtrl,
                     I_AlarmC := "FALSE",
                     I_AlarmD := "FALSE",
                     I_SafetyOk := "FALSE",
                     I_Service := "FALSE",
                     I_Spare1 := "FALSE",
                     I_Spare2 := "FALSE",
                     I_Spare3 := "FALSE",
                     I_Spare4 := "FALSE",
                     I_Spare5 := "FALSE",
                     I_Spare6 := "FALSE",
                     I_Spare7 := "FALSE",
                     I_Spare8 := "FALSE",
                     I_Spare9 := "FALSE",
                     I_Spare10 := "FALSE",
                     I_Spare11 := "FALSE",
                     I_Spare12 := "FALSE",
                     I_Spare13 := "FALSE",
                     I_Spare14 := "FALSE",
                     H_IAnim => #"H_GBHoist2Pos2S-C".H_LSpdDetSetCtrlIAnim[1].H_DWord);
   END_IF;
END_REGION

REGION Network 22: **** 4.6 - Machine status - Indications **** ContBypassOverTravelSetIAnim
   // Contactor overtravel bypass Set animation
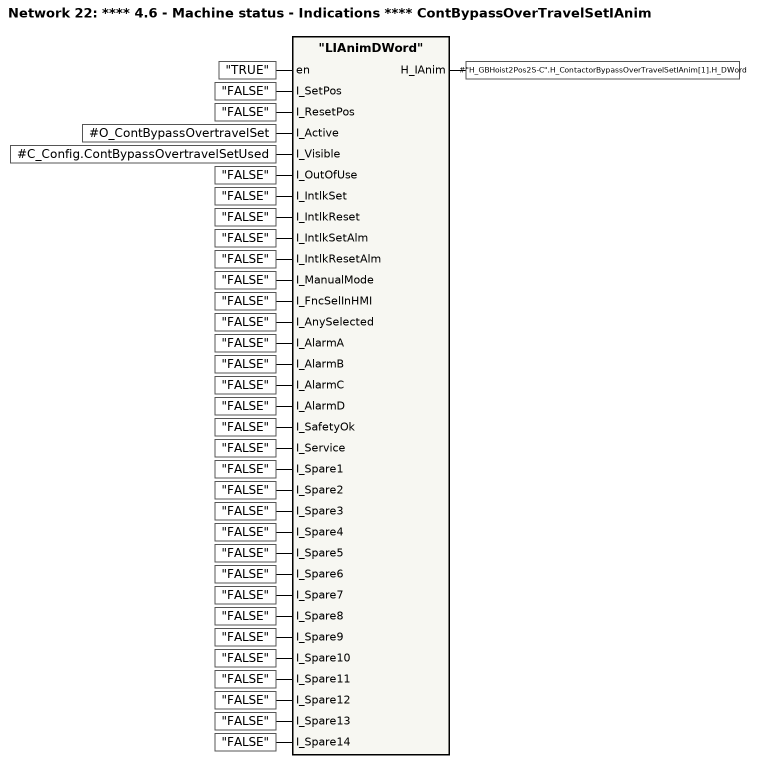
   IF "TRUE" THEN
       "LIAnimDWord"(I_SetPos := "FALSE",
                     I_ResetPos := "FALSE",
                     I_Active := #O_ContBypassOvertravelSet,
                     I_Visible := #C_Config.ContBypassOvertravelSetUsed,
                     I_OutOfUse := "FALSE",
                     I_IntlkSet := "FALSE",
                     I_IntlkReset := "FALSE",
                     I_IntlkSetAlm := "FALSE",
                     I_IntlkResetAlm := "FALSE",
                     I_ManualMode := "FALSE",
                     I_FncSelInHMI := "FALSE",
                     I_AnySelected := "FALSE",
                     I_AlarmA := "FALSE",
                     I_AlarmB := "FALSE",
                     I_AlarmC := "FALSE",
                     I_AlarmD := "FALSE",
                     I_SafetyOk := "FALSE",
                     I_Service := "FALSE",
                     I_Spare1 := "FALSE",
                     I_Spare2 := "FALSE",
                     I_Spare3 := "FALSE",
                     I_Spare4 := "FALSE",
                     I_Spare5 := "FALSE",
                     I_Spare6 := "FALSE",
                     I_Spare7 := "FALSE",
                     I_Spare8 := "FALSE",
                     I_Spare9 := "FALSE",
                     I_Spare10 := "FALSE",
                     I_Spare11 := "FALSE",
                     I_Spare12 := "FALSE",
                     I_Spare13 := "FALSE",
                     I_Spare14 := "FALSE",
                     H_IAnim => #"H_GBHoist2Pos2S-C".H_ContactorBypassOverTravelSetIAnim[1].H_DWord);
   END_IF;
END_REGION

REGION Network 23: **** 4.6 - Machine status - Indications **** LSpeedDetResIAnim
   // Low speed detector Reset animation
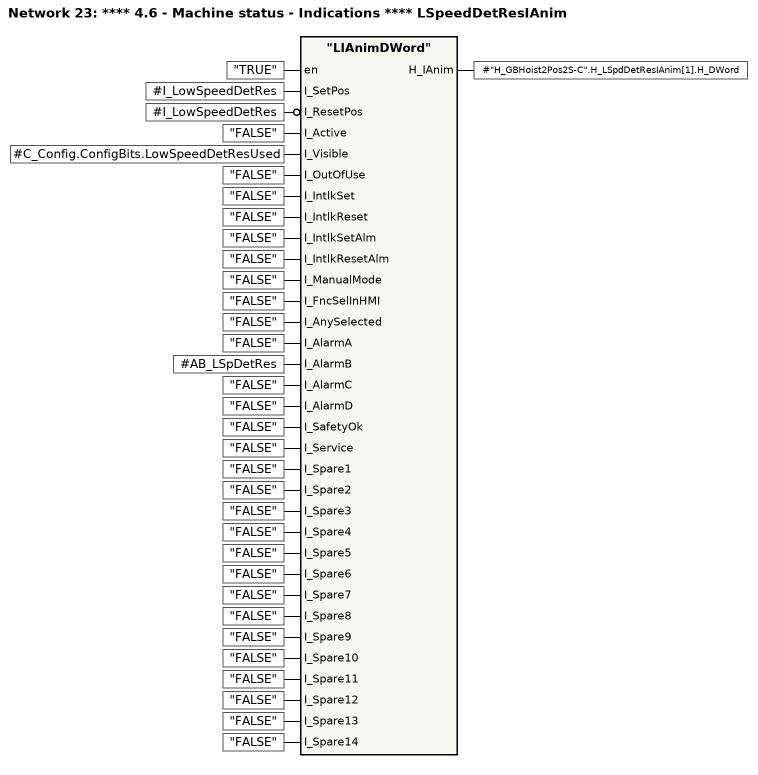
   IF "TRUE" THEN
       "LIAnimDWord"(I_SetPos := #I_LowSpeedDetRes,
                     I_ResetPos := NOT #I_LowSpeedDetRes,
                     I_Active := "FALSE",
                     I_Visible := #C_Config.ConfigBits.LowSpeedDetResUsed,
                     I_OutOfUse := "FALSE",
                     I_IntlkSet := "FALSE",
                     I_IntlkReset := "FALSE",
                     I_IntlkSetAlm := "FALSE",
                     I_IntlkResetAlm := "FALSE",
                     I_ManualMode := "FALSE",
                     I_FncSelInHMI := "FALSE",
                     I_AnySelected := "FALSE",
                     I_AlarmA := "FALSE",
                     I_AlarmB := #AB_LSpDetRes,
                     I_AlarmC := "FALSE",
                     I_AlarmD := "FALSE",
                     I_SafetyOk := "FALSE",
                     I_Service := "FALSE",
                     I_Spare1 := "FALSE",
                     I_Spare2 := "FALSE",
                     I_Spare3 := "FALSE",
                     I_Spare4 := "FALSE",
                     I_Spare5 := "FALSE",
                     I_Spare6 := "FALSE",
                     I_Spare7 := "FALSE",
                     I_Spare8 := "FALSE",
                     I_Spare9 := "FALSE",
                     I_Spare10 := "FALSE",
                     I_Spare11 := "FALSE",
                     I_Spare12 := "FALSE",
                     I_Spare13 := "FALSE",
                     I_Spare14 := "FALSE",
                     H_IAnim => #"H_GBHoist2Pos2S-C".H_LSpdDetResIAnim[1].H_DWord);
   END_IF;
END_REGION

REGION Network 24: **** 4.6 - Machine status - Indications **** LSpeedDetResCtrlIAnim
   // Low speed detector Control animation
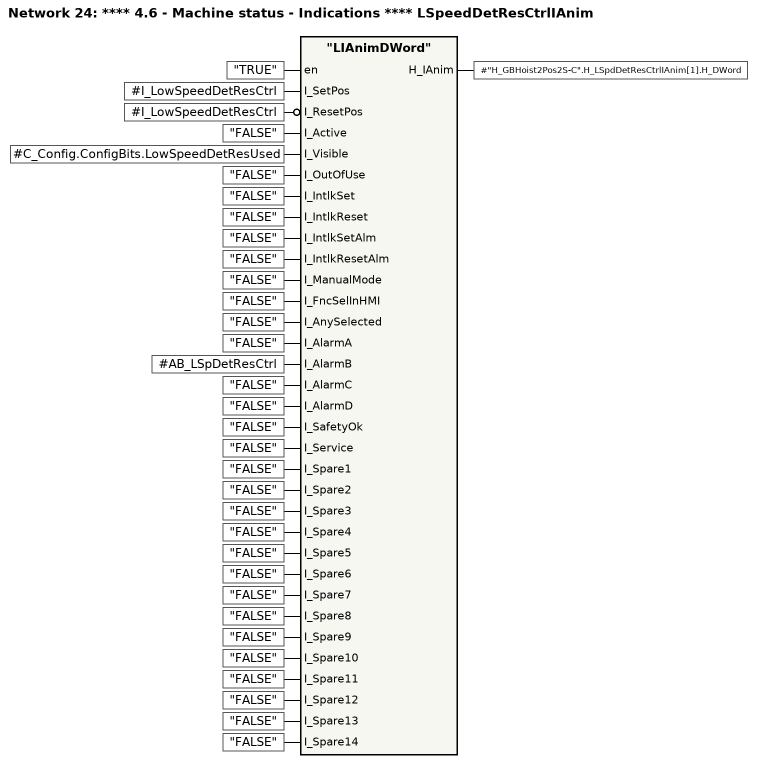
   IF "TRUE" THEN
       "LIAnimDWord"(I_SetPos := #I_LowSpeedDetResCtrl,
                     I_ResetPos := NOT #I_LowSpeedDetResCtrl,
                     I_Active := "FALSE",
                     I_Visible := #C_Config.ConfigBits.LowSpeedDetResUsed,
                     I_OutOfUse := "FALSE",
                     I_IntlkSet := "FALSE",
                     I_IntlkReset := "FALSE",
                     I_IntlkSetAlm := "FALSE",
                     I_IntlkResetAlm := "FALSE",
                     I_ManualMode := "FALSE",
                     I_FncSelInHMI := "FALSE",
                     I_AnySelected := "FALSE",
                     I_AlarmA := "FALSE",
                     I_AlarmB := #AB_LSpDetResCtrl,
                     I_AlarmC := "FALSE",
                     I_AlarmD := "FALSE",
                     I_SafetyOk := "FALSE",
                     I_Service := "FALSE",
                     I_Spare1 := "FALSE",
                     I_Spare2 := "FALSE",
                     I_Spare3 := "FALSE",
                     I_Spare4 := "FALSE",
                     I_Spare5 := "FALSE",
                     I_Spare6 := "FALSE",
                     I_Spare7 := "FALSE",
                     I_Spare8 := "FALSE",
                     I_Spare9 := "FALSE",
                     I_Spare10 := "FALSE",
                     I_Spare11 := "FALSE",
                     I_Spare12 := "FALSE",
                     I_Spare13 := "FALSE",
                     I_Spare14 := "FALSE",
                     H_IAnim => #"H_GBHoist2Pos2S-C".H_LSpdDetResCtrlIAnim[1].H_DWord);
   END_IF;
END_REGION

REGION Network 25: **** 4.6 - Machine status - Indications **** StopDetResIAnim
   // Stop detector Reset animation
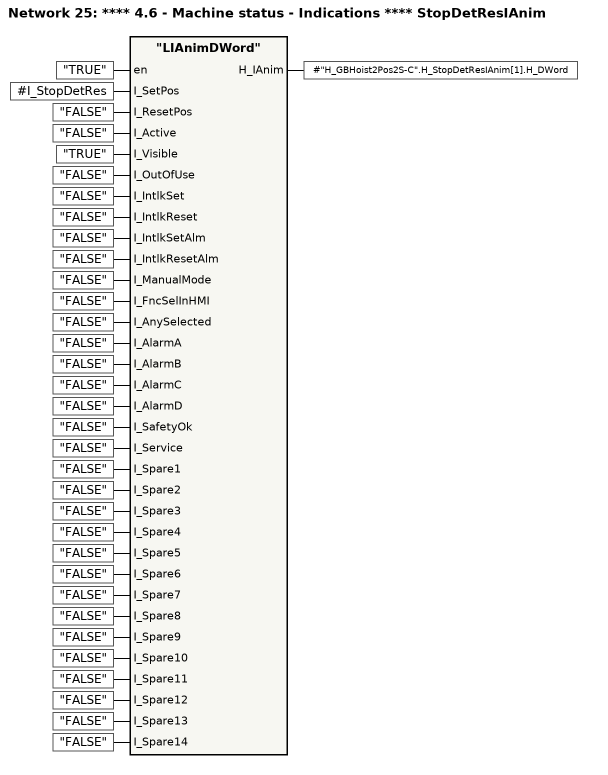
   IF "TRUE" THEN
       "LIAnimDWord"(I_SetPos := #I_StopDetRes,
                     I_ResetPos := "FALSE",
                     I_Active := "FALSE",
                     I_Visible := "TRUE",
                     I_OutOfUse := "FALSE",
                     I_IntlkSet := "FALSE",
                     I_IntlkReset := "FALSE",
                     I_IntlkSetAlm := "FALSE",
                     I_IntlkResetAlm := "FALSE",
                     I_ManualMode := "FALSE",
                     I_FncSelInHMI := "FALSE",
                     I_AnySelected := "FALSE",
                     I_AlarmA := "FALSE",
                     I_AlarmB := "FALSE",
                     I_AlarmC := "FALSE",
                     I_AlarmD := "FALSE",
                     I_SafetyOk := "FALSE",
                     I_Service := "FALSE",
                     I_Spare1 := "FALSE",
                     I_Spare2 := "FALSE",
                     I_Spare3 := "FALSE",
                     I_Spare4 := "FALSE",
                     I_Spare5 := "FALSE",
                     I_Spare6 := "FALSE",
                     I_Spare7 := "FALSE",
                     I_Spare8 := "FALSE",
                     I_Spare9 := "FALSE",
                     I_Spare10 := "FALSE",
                     I_Spare11 := "FALSE",
                     I_Spare12 := "FALSE",
                     I_Spare13 := "FALSE",
                     I_Spare14 := "FALSE",
                     H_IAnim => #"H_GBHoist2Pos2S-C".H_StopDetResIAnim[1].H_DWord);
   END_IF;
END_REGION

REGION Network 26: **** 4.6 - Machine status - Indications **** ContBypassOverTravelResIAnim
   // Contactor overtravel bypass Res animation
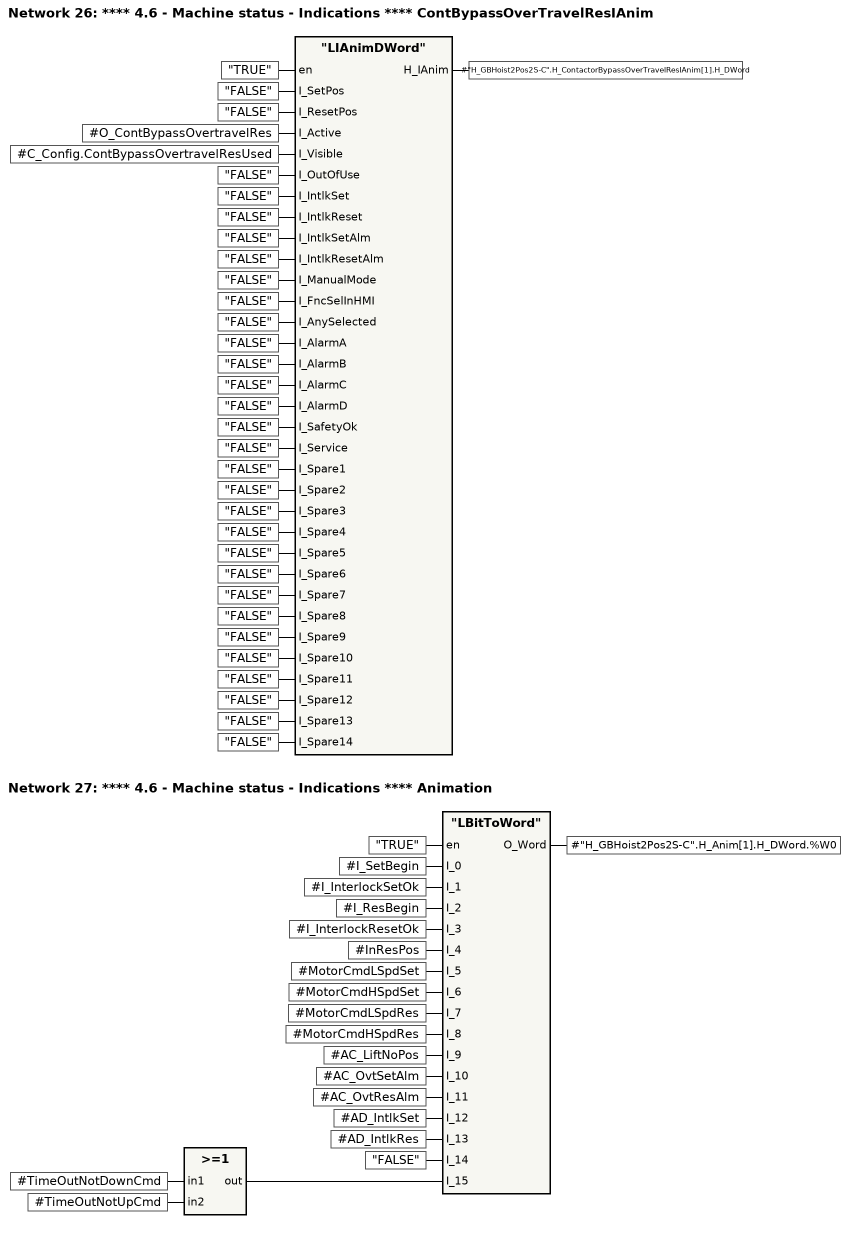
   IF "TRUE" THEN
       "LIAnimDWord"(I_SetPos := "FALSE",
                     I_ResetPos := "FALSE",
                     I_Active := #O_ContBypassOvertravelRes,
                     I_Visible := #C_Config.ContBypassOvertravelResUsed,
                     I_OutOfUse := "FALSE",
                     I_IntlkSet := "FALSE",
                     I_IntlkReset := "FALSE",
                     I_IntlkSetAlm := "FALSE",
                     I_IntlkResetAlm := "FALSE",
                     I_ManualMode := "FALSE",
                     I_FncSelInHMI := "FALSE",
                     I_AnySelected := "FALSE",
                     I_AlarmA := "FALSE",
                     I_AlarmB := "FALSE",
                     I_AlarmC := "FALSE",
                     I_AlarmD := "FALSE",
                     I_SafetyOk := "FALSE",
                     I_Service := "FALSE",
                     I_Spare1 := "FALSE",
                     I_Spare2 := "FALSE",
                     I_Spare3 := "FALSE",
                     I_Spare4 := "FALSE",
                     I_Spare5 := "FALSE",
                     I_Spare6 := "FALSE",
                     I_Spare7 := "FALSE",
                     I_Spare8 := "FALSE",
                     I_Spare9 := "FALSE",
                     I_Spare10 := "FALSE",
                     I_Spare11 := "FALSE",
                     I_Spare12 := "FALSE",
                     I_Spare13 := "FALSE",
                     I_Spare14 := "FALSE",
                     H_IAnim => #"H_GBHoist2Pos2S-C".H_ContactorBypassOverTravelResIAnim[1].H_DWord);
   END_IF;
END_REGION

REGION Network 27: **** 4.6 - Machine status - Indications **** Animation
   // Animation for HMI
   IF "TRUE" THEN
       "LBitToWord"(I_0 := #I_SetBegin,
                    I_1 := #I_InterlockSetOk,
                    I_2 := #I_ResBegin,
                    I_3 := #I_InterlockResetOk,
                    I_4 := #InResPos,
                    I_5 := #MotorCmdLSpdSet,
                    I_6 := #MotorCmdHSpdSet,
                    I_7 := #MotorCmdLSpdRes,
                    I_8 := #MotorCmdHSpdRes,
                    I_9 := #AC_LiftNoPos,
                    I_10 := #AC_OvtSetAlm,
                    I_11 := #AC_OvtResAlm,
                    I_12 := #AD_IntlkSet,
                    I_13 := #AD_IntlkRes,
                    I_14 := "FALSE",
                    I_15 := #TimeOutNotDownCmd OR #TimeOutNotUpCmd,
                    O_Word => #"H_GBHoist2Pos2S-C".H_Anim[1].H_DWord.%W0);
   END_IF;
END_REGION

REGION Network 28: **** 4.6 - Machine status - Indications **** Animation
   // Animation for HMI
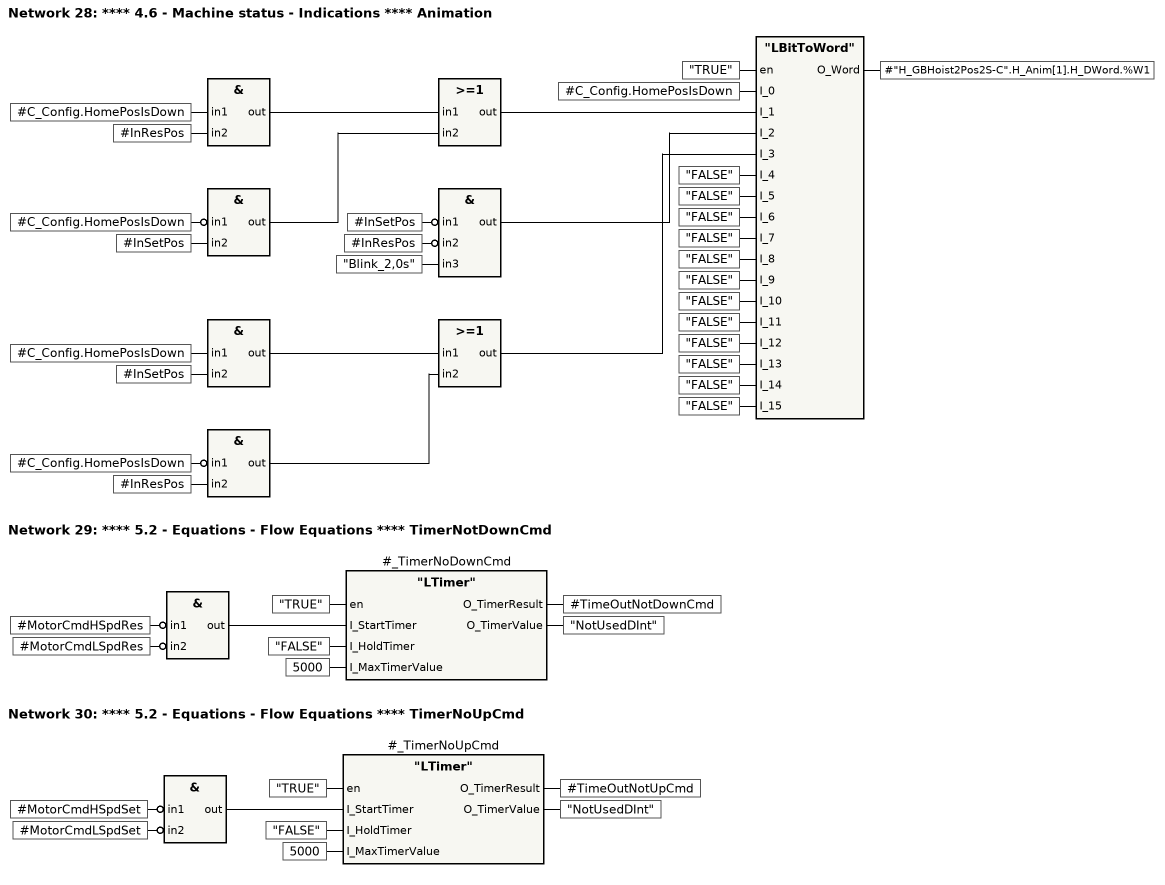
   IF "TRUE" THEN
       "LBitToWord"(I_0 := #C_Config.HomePosIsDown,
                    I_1 := (#C_Config.HomePosIsDown AND #InResPos) OR (NOT #C_Config.HomePosIsDown AND #InSetPos),
                    I_2 := NOT #InSetPos AND NOT #InResPos AND "Blink_2,0s",
                    I_3 := (#C_Config.HomePosIsDown AND #InSetPos) OR (NOT #C_Config.HomePosIsDown AND #InResPos),
                    I_4 := "FALSE",
                    I_5 := "FALSE",
                    I_6 := "FALSE",
                    I_7 := "FALSE",
                    I_8 := "FALSE",
                    I_9 := "FALSE",
                    I_10 := "FALSE",
                    I_11 := "FALSE",
                    I_12 := "FALSE",
                    I_13 := "FALSE",
                    I_14 := "FALSE",
                    I_15 := "FALSE",
                    O_Word => #"H_GBHoist2Pos2S-C".H_Anim[1].H_DWord.%W1);
   END_IF;
END_REGION

REGION Network 29: **** 5.2 - Equations - Flow Equations **** TimerNotDownCmd
   // Timer, no down (Reset) movement, the hoist must not move in the opposite direction before time is out.
   IF "TRUE" THEN
       #_TimerNoDownCmd(I_StartTimer := NOT #MotorCmdHSpdRes AND NOT #MotorCmdLSpdRes,   // "LTimer"
                        I_HoldTimer := "FALSE",
                        I_MaxTimerValue := 5000,
                        O_TimerResult => #TimeOutNotDownCmd,
                        O_TimerValue => "NotUsedDInt");
   END_IF;
END_REGION

REGION Network 30: **** 5.2 - Equations - Flow Equations **** TimerNoUpCmd
   // Timer, no up (Set) movement, the hoist must not move in the opposite direction 
   // before time is up.
   IF "TRUE" THEN
       #_TimerNoUpCmd(I_StartTimer := NOT #MotorCmdHSpdSet AND NOT #MotorCmdLSpdSet,   // "LTimer"
                      I_HoldTimer := "FALSE",
                      I_MaxTimerValue := 5000,
                      O_TimerResult => #TimeOutNotUpCmd,
                      O_TimerValue => "NotUsedDInt");
   END_IF;
END_REGION

REGION Network 31: **** 5.2 - Equations - Flow Equations **** HighSpeedMem
   // High speed memory
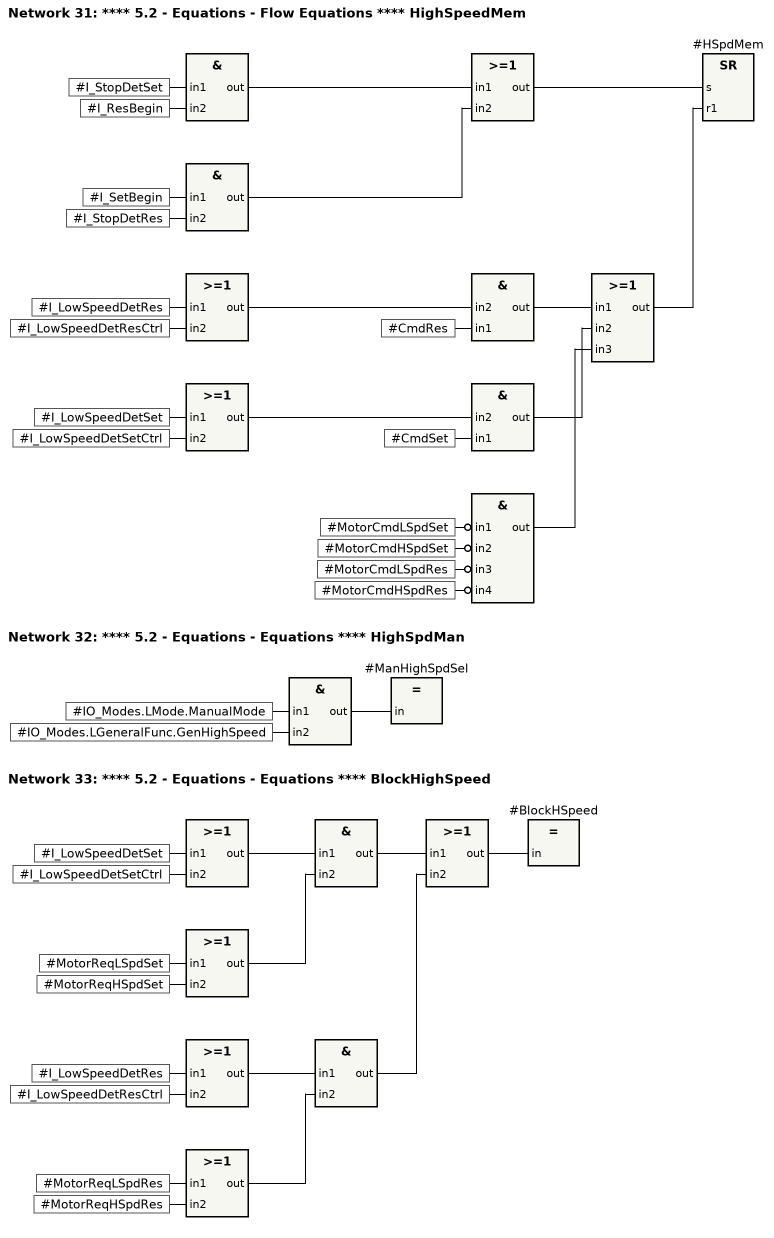
   IF (#I_StopDetSet AND #I_ResBegin) OR (#I_SetBegin AND #I_StopDetRes) THEN
       #HSpdMem := TRUE;   // SR flip-flop
   END_IF;
   IF ((#I_LowSpeedDetRes OR #I_LowSpeedDetResCtrl) AND #CmdRes) OR ((#I_LowSpeedDetSet OR #I_LowSpeedDetSetCtrl) AND #CmdSet) OR (NOT #MotorCmdLSpdSet AND NOT #MotorCmdHSpdSet AND NOT #MotorCmdLSpdRes AND NOT #MotorCmdHSpdRes) THEN
       #HSpdMem := FALSE;
   END_IF;
END_REGION

REGION Network 32: **** 5.2 - Equations - Equations **** HighSpdMan
   // Cmd summary high speed in manual
   #ManHighSpdSel := #IO_Modes.LMode.ManualMode AND #IO_Modes.LGeneralFunc.GenHighSpeed;
END_REGION

REGION Network 33: **** 5.2 - Equations - Equations **** BlockHighSpeed
   // Block High Speed
   #BlockHSpeed := ((#I_LowSpeedDetSet OR #I_LowSpeedDetSetCtrl) AND (#MotorReqLSpdSet OR #MotorReqHSpdSet)) OR ((#I_LowSpeedDetRes OR #I_LowSpeedDetResCtrl) AND (#MotorReqLSpdRes OR #MotorReqHSpdRes));
END_REGION

REGION Network 34: **** 5.2 - Equations - Equations **** LowSpeedSet
   // Motor Command Low Speed Set (up)
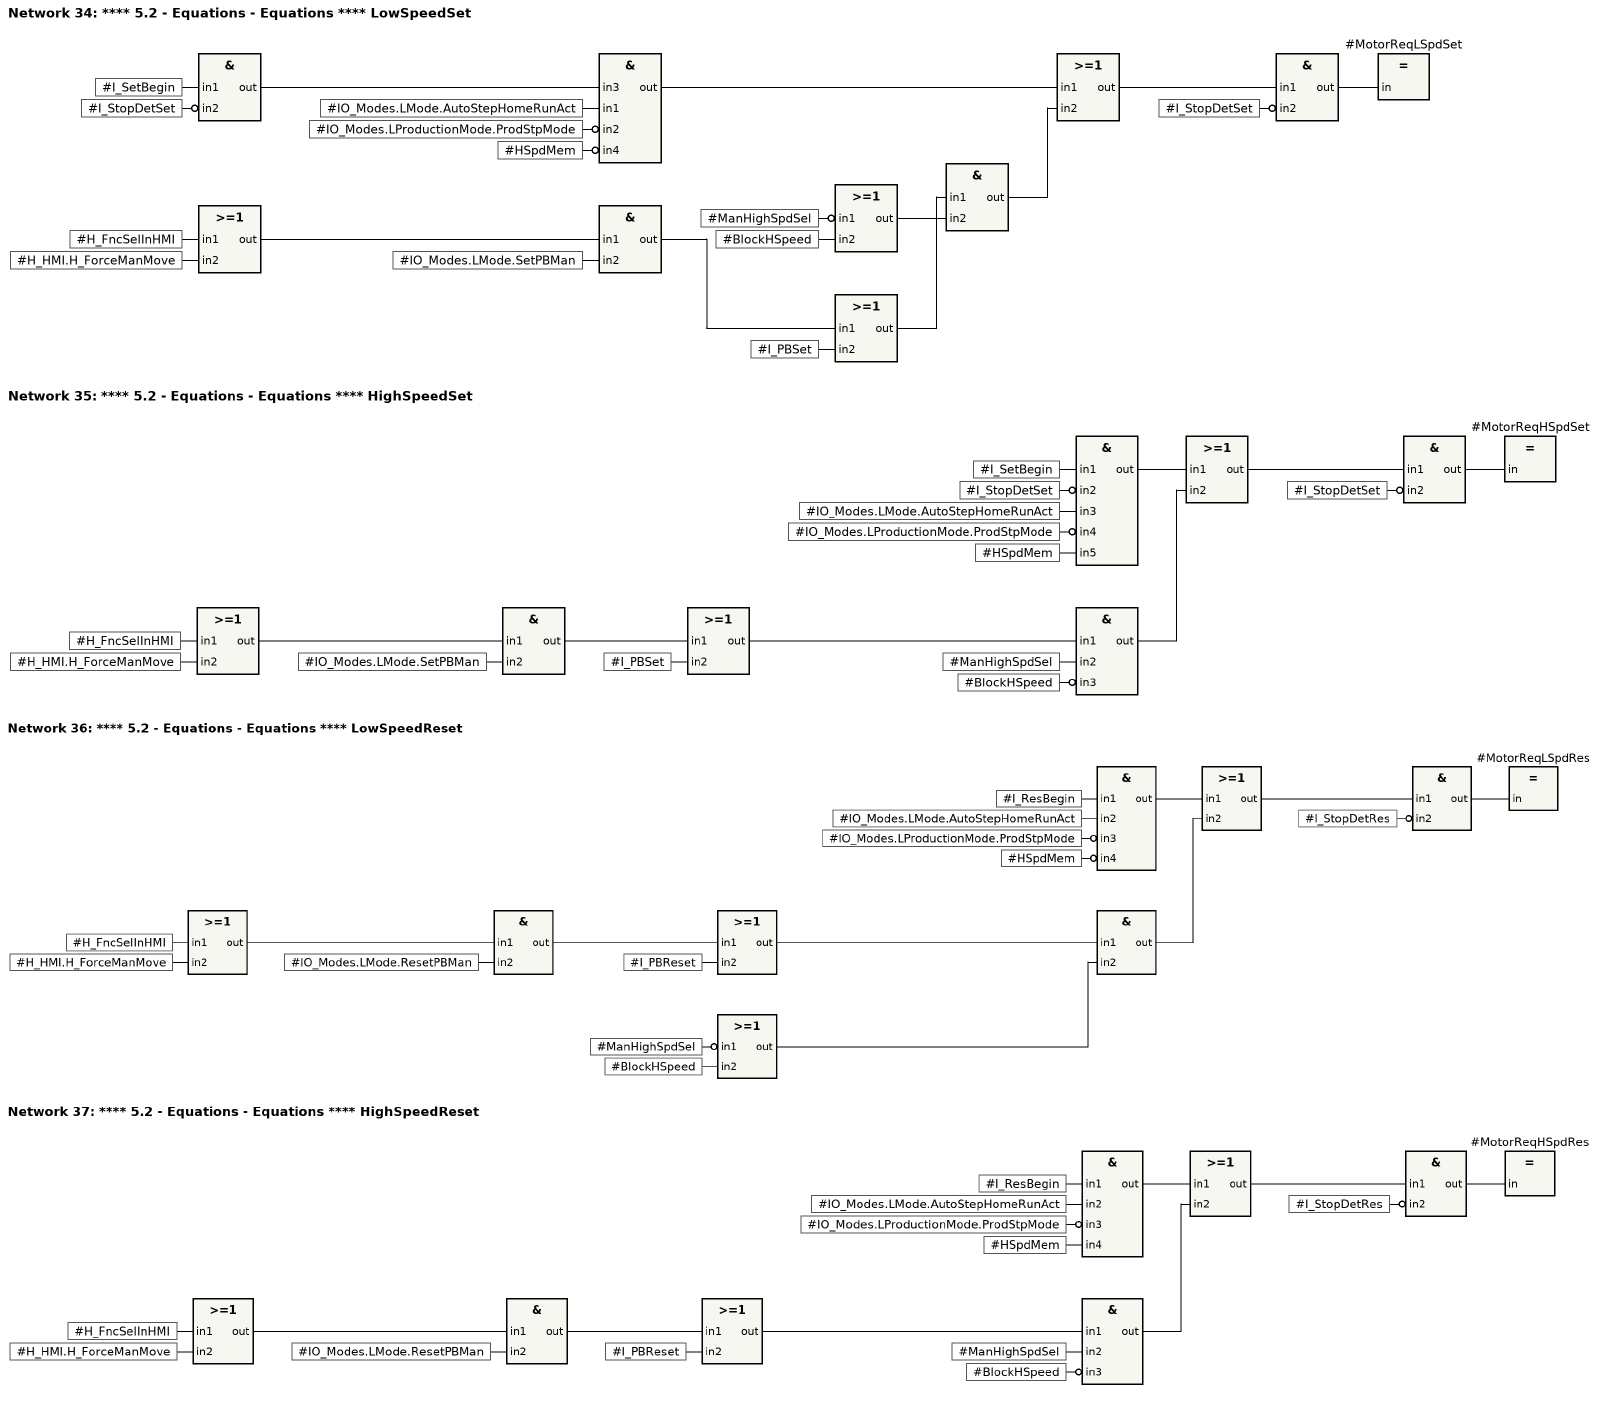
   #MotorReqLSpdSet := ((#I_SetBegin AND NOT #I_StopDetSet AND #IO_Modes.LMode.AutoStepHomeRunAct AND NOT #IO_Modes.LProductionMode.ProdStpMode AND NOT #HSpdMem) OR ((((#H_FncSelInHMI OR #H_HMI.H_ForceManMove) AND #IO_Modes.LMode.SetPBMan) OR #I_PBSet) AND (NOT #ManHighSpdSel OR #BlockHSpeed))) AND NOT #I_StopDetSet;
END_REGION

REGION Network 35: **** 5.2 - Equations - Equations **** HighSpeedSet
   // Motor command high Speed Set (up)
   #MotorReqHSpdSet := ((#I_SetBegin AND NOT #I_StopDetSet AND #IO_Modes.LMode.AutoStepHomeRunAct AND NOT #IO_Modes.LProductionMode.ProdStpMode AND #HSpdMem) OR ((((#H_FncSelInHMI OR #H_HMI.H_ForceManMove) AND #IO_Modes.LMode.SetPBMan) OR #I_PBSet) AND #ManHighSpdSel AND NOT #BlockHSpeed)) AND NOT #I_StopDetSet;
END_REGION

REGION Network 36: **** 5.2 - Equations - Equations **** LowSpeedReset
   // Motor Command Low Speed Reset (down)
   #MotorReqLSpdRes := ((#I_ResBegin AND #IO_Modes.LMode.AutoStepHomeRunAct AND NOT #IO_Modes.LProductionMode.ProdStpMode AND NOT #HSpdMem) OR ((((#H_FncSelInHMI OR #H_HMI.H_ForceManMove) AND #IO_Modes.LMode.ResetPBMan) OR #I_PBReset) AND (NOT #ManHighSpdSel OR #BlockHSpeed))) AND NOT #I_StopDetRes;
END_REGION

REGION Network 37: **** 5.2 - Equations - Equations **** HighSpeedReset
   // Motor command high speed Reset (down)
   #MotorReqHSpdRes := ((#I_ResBegin AND #IO_Modes.LMode.AutoStepHomeRunAct AND NOT #IO_Modes.LProductionMode.ProdStpMode AND #HSpdMem) OR ((((#H_FncSelInHMI OR #H_HMI.H_ForceManMove) AND #IO_Modes.LMode.ResetPBMan) OR #I_PBReset) AND #ManHighSpdSel AND NOT #BlockHSpeed)) AND NOT #I_StopDetRes;
END_REGION

REGION Network 38: **** 5.2 - Equations - Equations **** Cmd LowSpeed Set
   // LowSpeed Set command
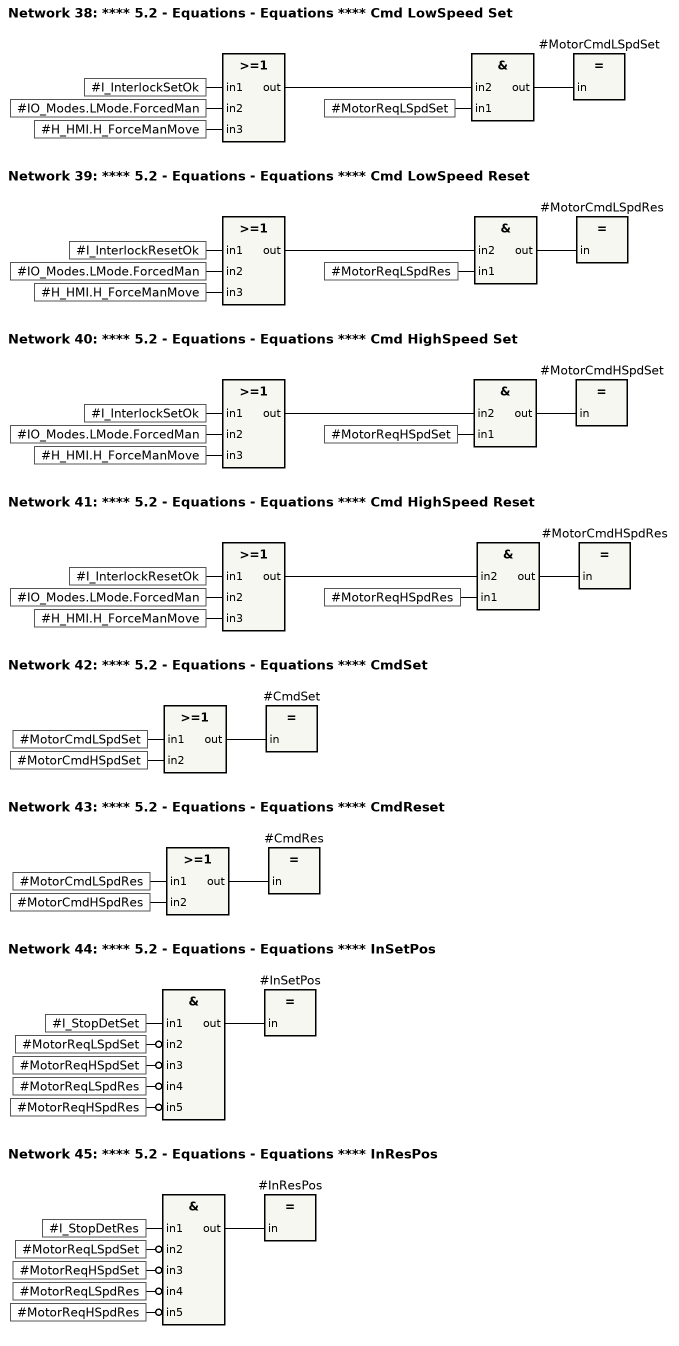
   #MotorCmdLSpdSet := (#I_InterlockSetOk OR #IO_Modes.LMode.ForcedMan OR #H_HMI.H_ForceManMove) AND #MotorReqLSpdSet;
END_REGION

REGION Network 39: **** 5.2 - Equations - Equations **** Cmd LowSpeed Reset
   // LowSpeed Reset command
   #MotorCmdLSpdRes := (#I_InterlockResetOk OR #IO_Modes.LMode.ForcedMan OR #H_HMI.H_ForceManMove) AND #MotorReqLSpdRes;
END_REGION

REGION Network 40: **** 5.2 - Equations - Equations **** Cmd HighSpeed Set
   // HighSpeedSet command
   #MotorCmdHSpdSet := (#I_InterlockSetOk OR #IO_Modes.LMode.ForcedMan OR #H_HMI.H_ForceManMove) AND #MotorReqHSpdSet;
END_REGION

REGION Network 41: **** 5.2 - Equations - Equations **** Cmd HighSpeed Reset
   // HighSpeedReset command
   #MotorCmdHSpdRes := (#I_InterlockResetOk OR #IO_Modes.LMode.ForcedMan OR #H_HMI.H_ForceManMove) AND #MotorReqHSpdRes;
END_REGION

REGION Network 42: **** 5.2 - Equations - Equations **** CmdSet
   // Set command
   #CmdSet := #MotorCmdLSpdSet OR #MotorCmdHSpdSet;
END_REGION

REGION Network 43: **** 5.2 - Equations - Equations **** CmdReset
   // Reset command
   #CmdRes := #MotorCmdLSpdRes OR #MotorCmdHSpdRes;
END_REGION

REGION Network 44: **** 5.2 - Equations - Equations **** InSetPos
   // In set Position
   #InSetPos := #I_StopDetSet AND NOT #MotorReqLSpdSet AND NOT #MotorReqHSpdSet AND NOT #MotorReqLSpdRes AND NOT #MotorReqHSpdRes;
END_REGION

REGION Network 45: **** 5.2 - Equations - Equations **** InResPos
   // In Reset Position
   #InResPos := #I_StopDetRes AND NOT #MotorReqLSpdSet AND NOT #MotorReqHSpdSet AND NOT #MotorReqLSpdRes AND NOT #MotorReqHSpdRes;
END_REGION

REGION Network 46: **** 7.3 - Submodule - Machine **** Motor loop
   // Motor loop
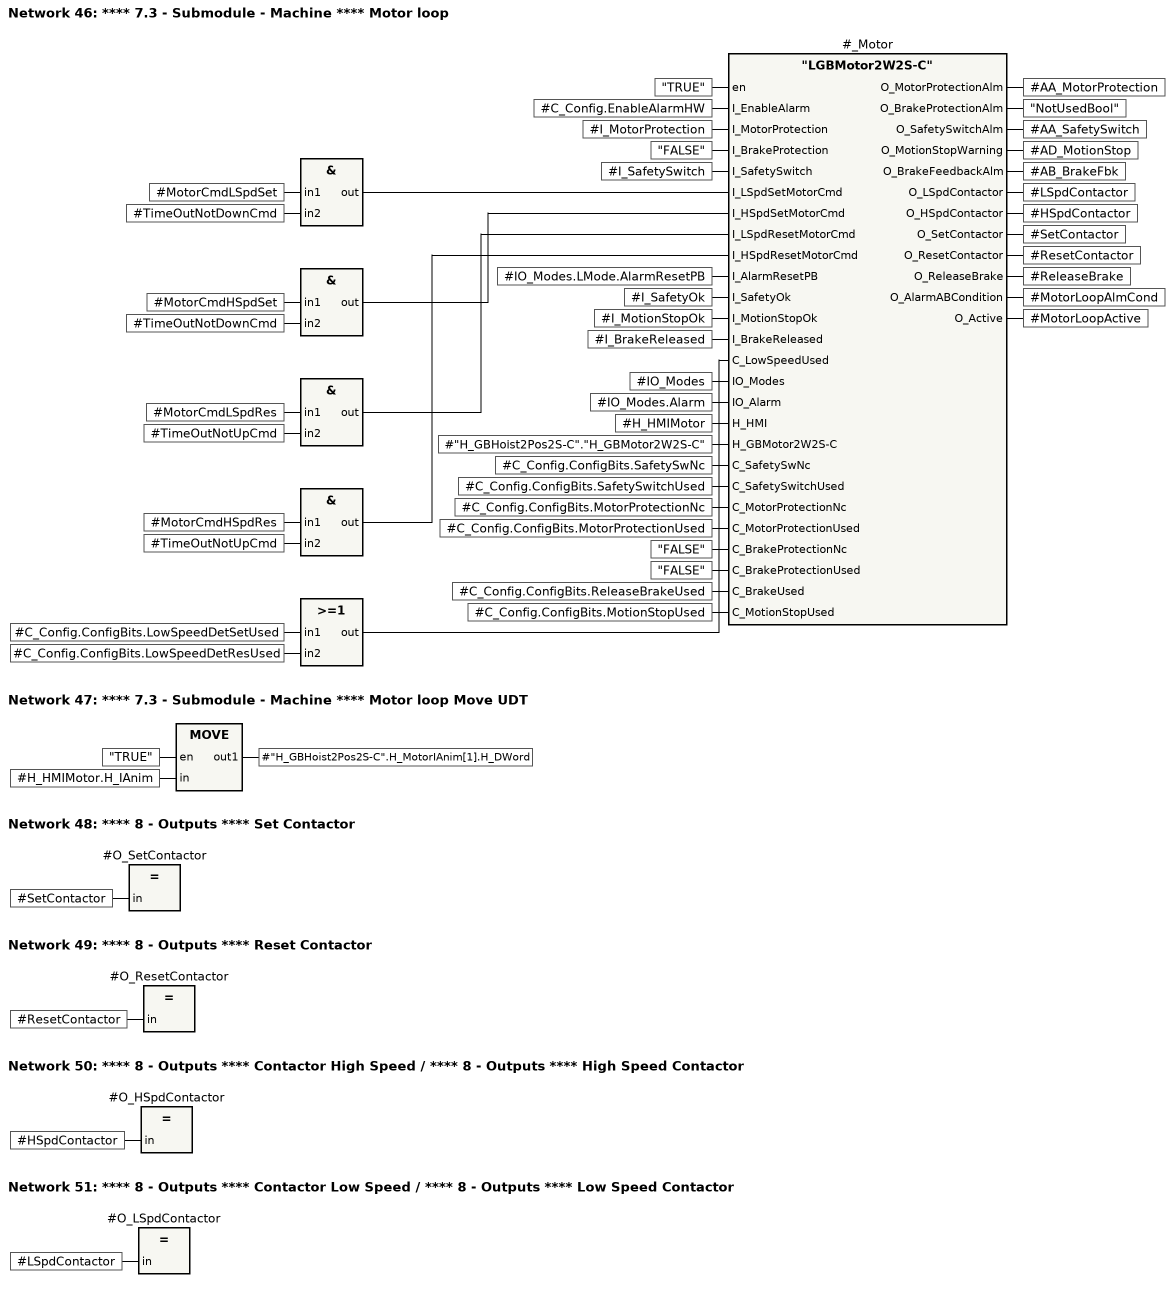
   IF "TRUE" THEN
       #_Motor(I_EnableAlarm := #C_Config.EnableAlarmHW,   // "LGBMotor2W2S-C"
               I_MotorProtection := #I_MotorProtection,
               I_BrakeProtection := "FALSE",
               I_SafetySwitch := #I_SafetySwitch,
               I_LSpdSetMotorCmd := #MotorCmdLSpdSet AND #TimeOutNotDownCmd,
               I_HSpdSetMotorCmd := #MotorCmdHSpdSet AND #TimeOutNotDownCmd,
               I_LSpdResetMotorCmd := #MotorCmdLSpdRes AND #TimeOutNotUpCmd,
               I_HSpdResetMotorCmd := #MotorCmdHSpdRes AND #TimeOutNotUpCmd,
               I_AlarmResetPB := #IO_Modes.LMode.AlarmResetPB,
               I_SafetyOk := #I_SafetyOk,
               I_MotionStopOk := #I_MotionStopOk,
               I_BrakeReleased := #I_BrakeReleased,
               C_LowSpeedUsed := #C_Config.ConfigBits.LowSpeedDetSetUsed OR #C_Config.ConfigBits.LowSpeedDetResUsed,
               IO_Modes := #IO_Modes,
               IO_Alarm := #IO_Modes.Alarm,
               H_HMI := #H_HMIMotor,
               "H_GBMotor2W2S-C" := #"H_GBHoist2Pos2S-C"."H_GBMotor2W2S-C",
               C_SafetySwNc := #C_Config.ConfigBits.SafetySwNc,
               C_SafetySwitchUsed := #C_Config.ConfigBits.SafetySwitchUsed,
               C_MotorProtectionNc := #C_Config.ConfigBits.MotorProtectionNc,
               C_MotorProtectionUsed := #C_Config.ConfigBits.MotorProtectionUsed,
               C_BrakeProtectionNc := "FALSE",
               C_BrakeProtectionUsed := "FALSE",
               C_BrakeUsed := #C_Config.ConfigBits.ReleaseBrakeUsed,
               C_MotionStopUsed := #C_Config.ConfigBits.MotionStopUsed,
               O_MotorProtectionAlm => #AA_MotorProtection,
               O_BrakeProtectionAlm => "NotUsedBool",
               O_SafetySwitchAlm => #AA_SafetySwitch,
               O_MotionStopWarning => #AD_MotionStop,
               O_BrakeFeedbackAlm => #AB_BrakeFbk,
               O_LSpdContactor => #LSpdContactor,
               O_HSpdContactor => #HSpdContactor,
               O_SetContactor => #SetContactor,
               O_ResetContactor => #ResetContactor,
               O_ReleaseBrake => #ReleaseBrake,
               O_AlarmABCondition => #MotorLoopAlmCond,
               O_Active => #MotorLoopActive);
   END_IF;
END_REGION

REGION Network 47: **** 7.3 - Submodule - Machine **** Motor loop Move UDT
   IF "TRUE" THEN #"H_GBHoist2Pos2S-C".H_MotorIAnim[1].H_DWord := #H_HMIMotor.H_IAnim; END_IF;
END_REGION

REGION Network 48: **** 8 - Outputs **** Set Contactor
   // Set Contactor
   #O_SetContactor := #SetContactor;
END_REGION

REGION Network 49: **** 8 - Outputs **** Reset Contactor
   // Reset Contactor
   #O_ResetContactor := #ResetContactor;
END_REGION

REGION Network 50: **** 8 - Outputs **** Contactor High Speed / **** 8 - Outputs **** High Speed Contactor
   // Contactor High Speed / High Speed Contactor
   #O_HSpdContactor := #HSpdContactor;
END_REGION

REGION Network 51: **** 8 - Outputs **** Contactor Low Speed / **** 8 - Outputs **** Low Speed Contactor
   // Contactor Low Speed / Low Speed Contactor
   #O_LSpdContactor := #LSpdContactor;
END_REGION

REGION Network 52: **** 8 - Outputs **** Release Brake
   // Release Brake
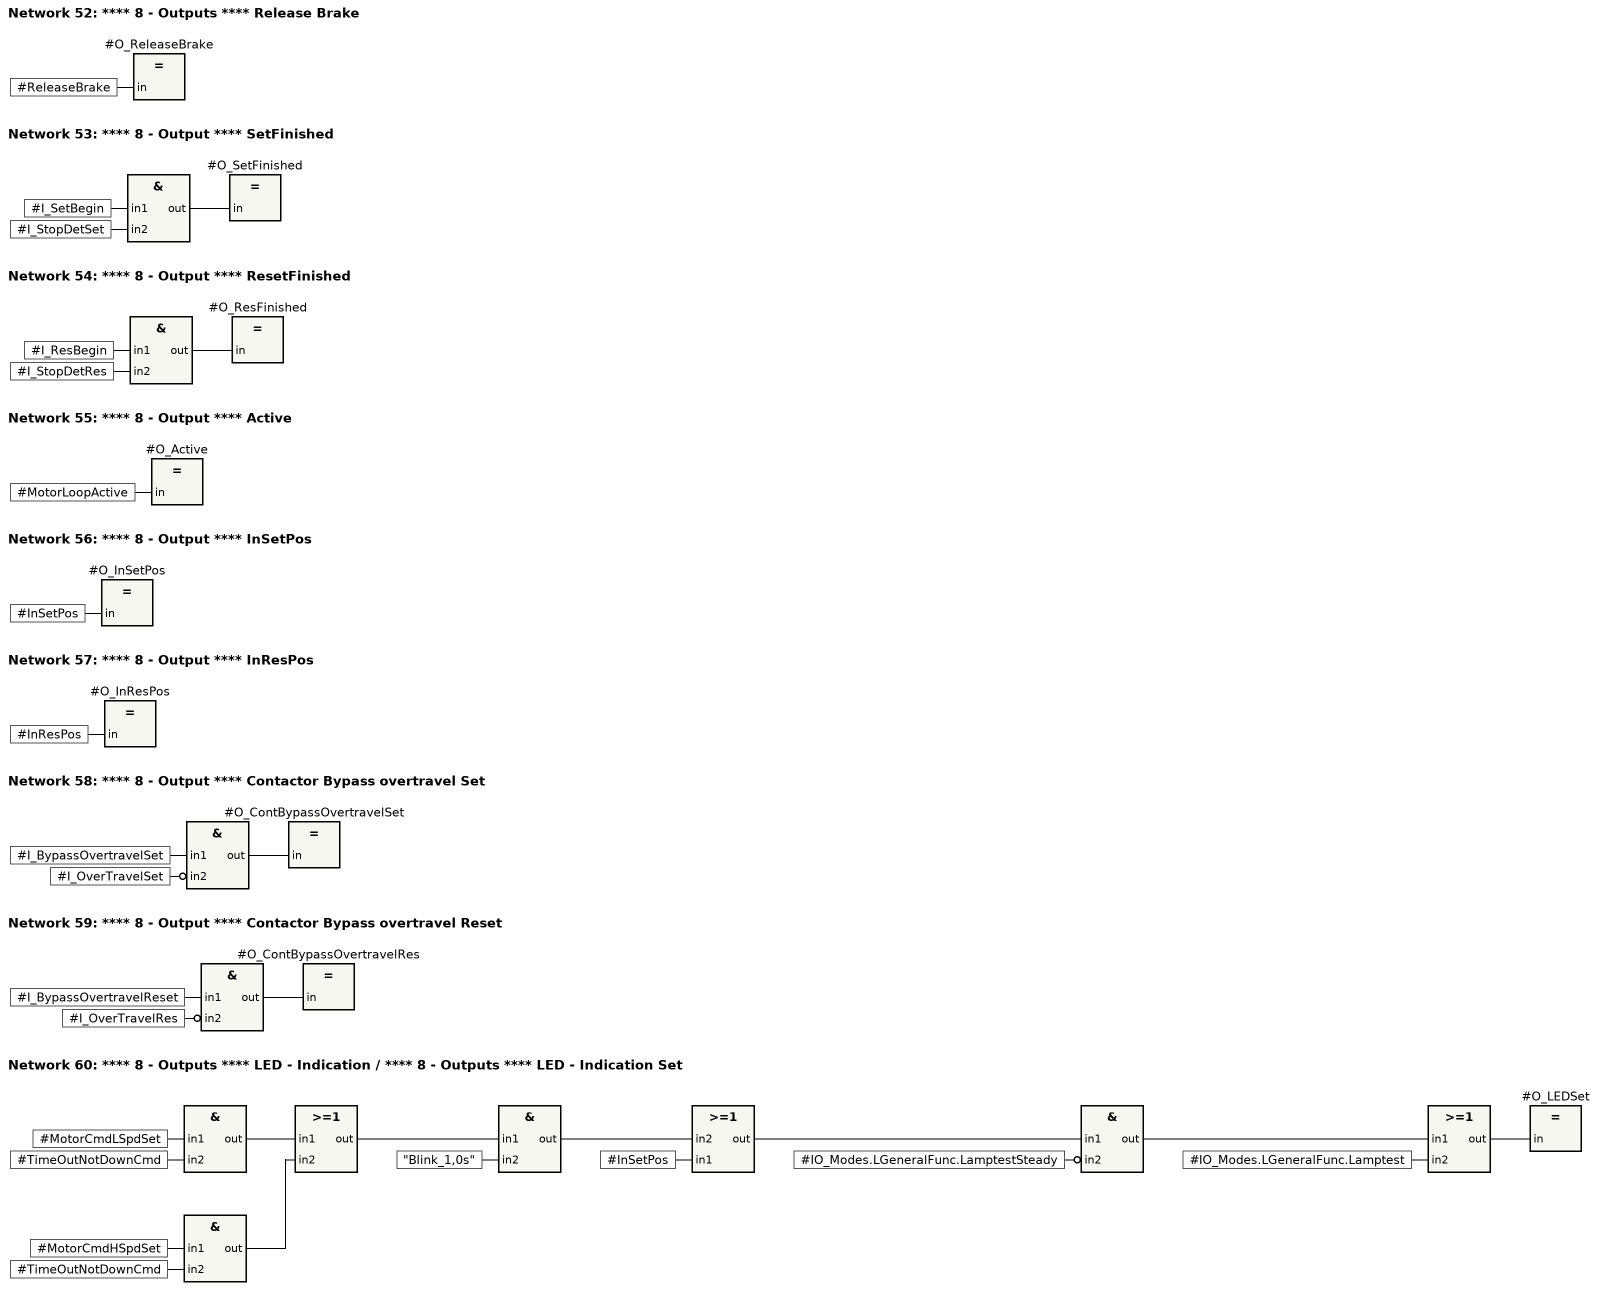
   #O_ReleaseBrake := #ReleaseBrake;
END_REGION

REGION Network 53: **** 8 - Output **** SetFinished
   // Handshake signal : Position Set (Up) Finished
   #O_SetFinished := #I_SetBegin AND #I_StopDetSet;
END_REGION

REGION Network 54: **** 8 - Output **** ResetFinished
   // Handshake signal : Position 2, Reset, Finished
   #O_ResFinished := #I_ResBegin AND #I_StopDetRes;
END_REGION

REGION Network 55: **** 8 - Output **** Active
   // Active
   #O_Active := #MotorLoopActive;
END_REGION

REGION Network 56: **** 8 - Output **** InSetPos
   // In Set Position
   #O_InSetPos := #InSetPos;
END_REGION

REGION Network 57: **** 8 - Output **** InResPos
   // In Reset Position
   #O_InResPos := #InResPos;
END_REGION

REGION Network 58: **** 8 - Output **** Contactor Bypass overtravel Set
   // Cmd Contactor bypass overtravel Set
   #O_ContBypassOvertravelSet := #I_BypassOvertravelSet AND NOT #I_OverTravelSet;
END_REGION

REGION Network 59: **** 8 - Output **** Contactor Bypass overtravel Reset
   // Cmd Contactor bypass overtravel Reset
   #O_ContBypassOvertravelRes := #I_BypassOvertravelReset AND NOT #I_OverTravelRes;
END_REGION

REGION Network 60: **** 8 - Outputs **** LED - Indication / **** 8 - Outputs **** LED - Indication Set
   // LED - Indication
   #O_LEDSet := (((((#MotorCmdLSpdSet AND #TimeOutNotDownCmd) OR (#MotorCmdHSpdSet AND #TimeOutNotDownCmd)) AND "Blink_1,0s") OR #InSetPos) AND NOT #IO_Modes.LGeneralFunc.LamptestSteady) OR #IO_Modes.LGeneralFunc.Lamptest;
END_REGION

REGION Network 61: **** 8 - Outputs **** LED - Indication / **** 8 - Outputs **** LED - Indication Reset
   // LED - Indication
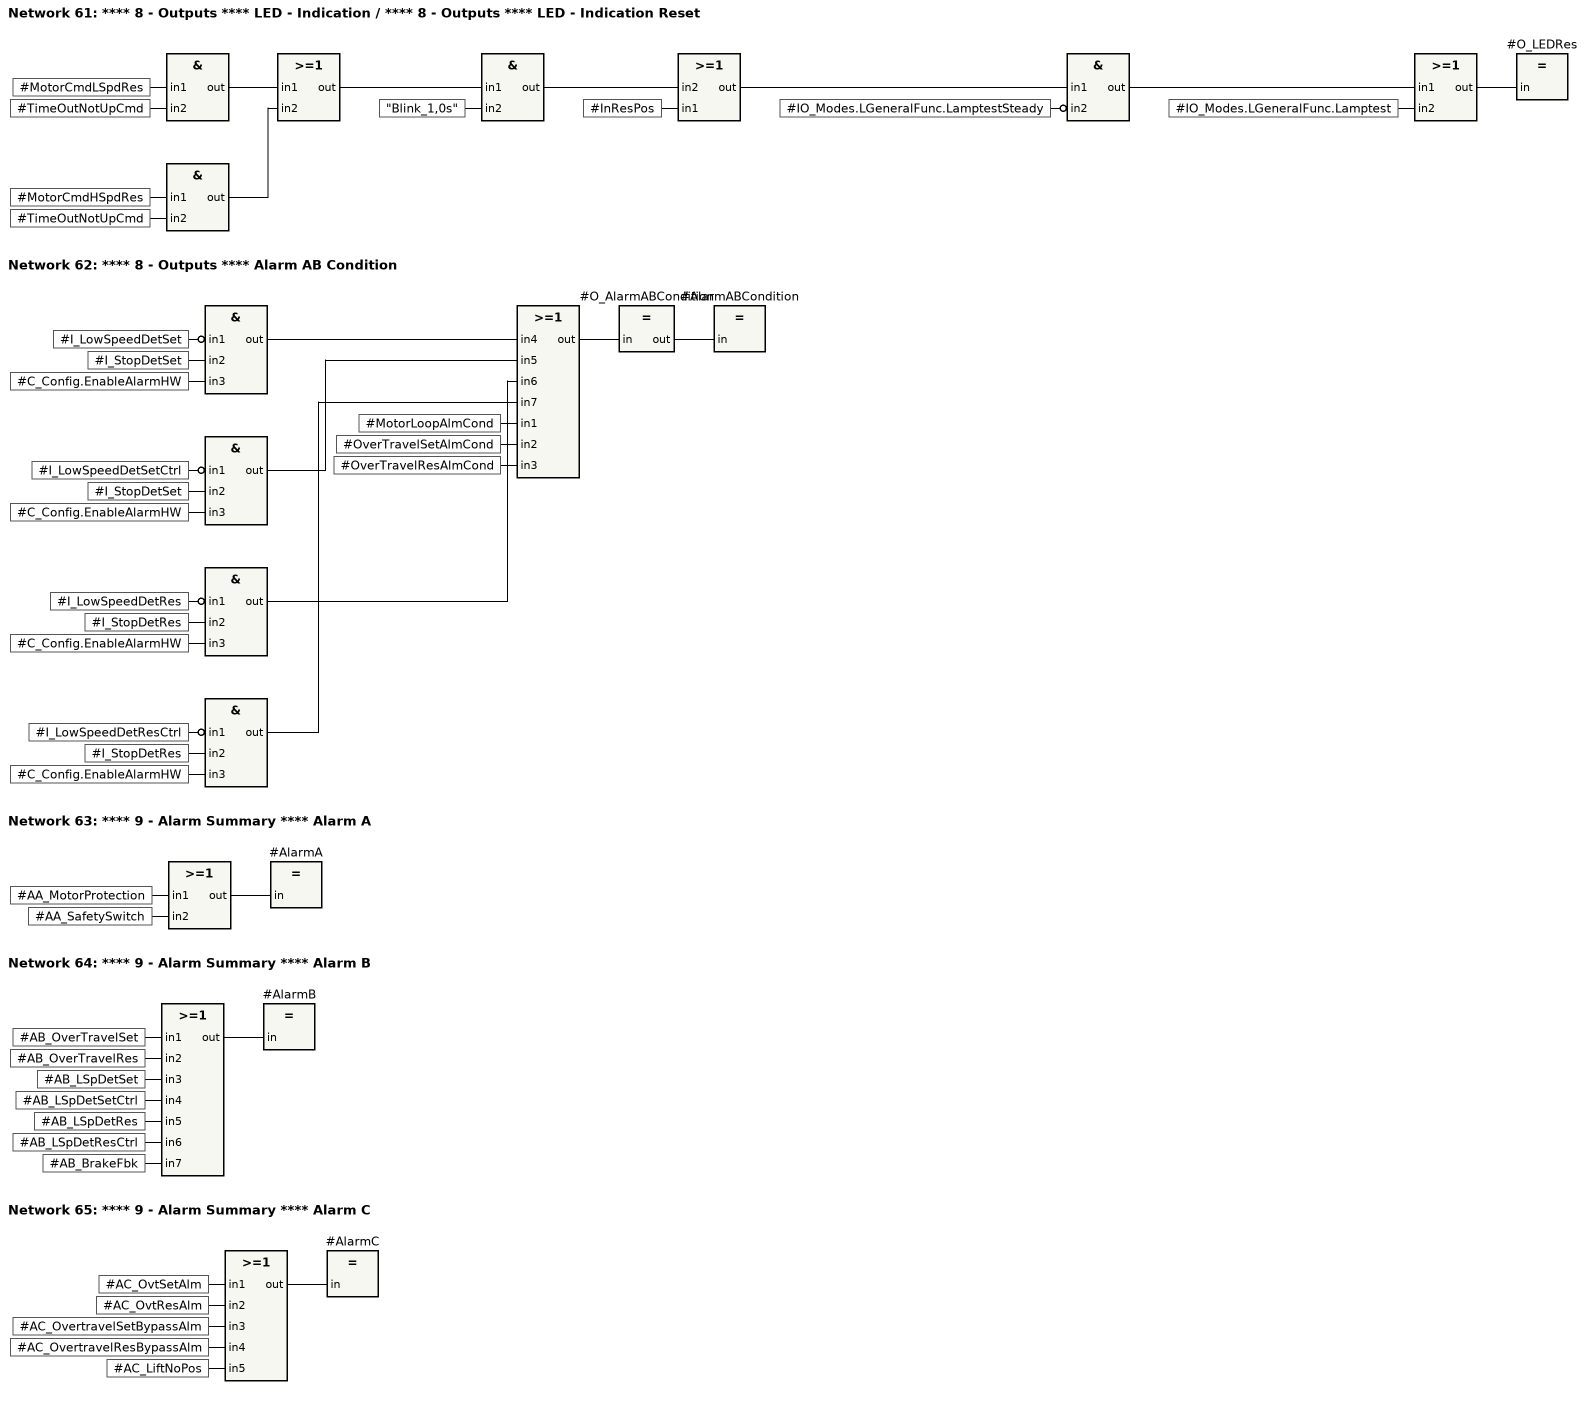
   #O_LEDRes := (((((#MotorCmdLSpdRes AND #TimeOutNotUpCmd) OR (#MotorCmdHSpdRes AND #TimeOutNotUpCmd)) AND "Blink_1,0s") OR #InResPos) AND NOT #IO_Modes.LGeneralFunc.LamptestSteady) OR #IO_Modes.LGeneralFunc.Lamptest;
END_REGION

REGION Network 62: **** 8 - Outputs **** Alarm AB Condition
   // Alarm AB Condition
   #O_AlarmABCondition := (NOT #I_LowSpeedDetSet AND #I_StopDetSet AND #C_Config.EnableAlarmHW) OR (NOT #I_LowSpeedDetSetCtrl AND #I_StopDetSet AND #C_Config.EnableAlarmHW) OR (NOT #I_LowSpeedDetRes AND #I_StopDetRes AND #C_Config.EnableAlarmHW) OR (NOT #I_LowSpeedDetResCtrl AND #I_StopDetRes AND #C_Config.EnableAlarmHW) OR #MotorLoopAlmCond OR #OverTravelSetAlmCond OR #OverTravelResAlmCond;
   #AlarmABCondition := #O_AlarmABCondition;
END_REGION

REGION Network 63: **** 9 - Alarm Summary **** Alarm A
   // Alarm A
   #AlarmA := #AA_MotorProtection OR #AA_SafetySwitch;
END_REGION

REGION Network 64: **** 9 - Alarm Summary **** Alarm B
   // Alarm B
   #AlarmB := #AB_OverTravelSet OR #AB_OverTravelRes OR #AB_LSpDetSet OR #AB_LSpDetSetCtrl OR #AB_LSpDetRes OR #AB_LSpDetResCtrl OR #AB_BrakeFbk;
END_REGION

REGION Network 65: **** 9 - Alarm Summary **** Alarm C
   // Alarm C
   #AlarmC := #AC_OvtSetAlm OR #AC_OvtResAlm OR #AC_OvertravelSetBypassAlm OR #AC_OvertravelResBypassAlm OR #AC_LiftNoPos;
END_REGION

REGION Network 66: **** 9 - Alarm Summary **** Alarm D
   // Alarm D
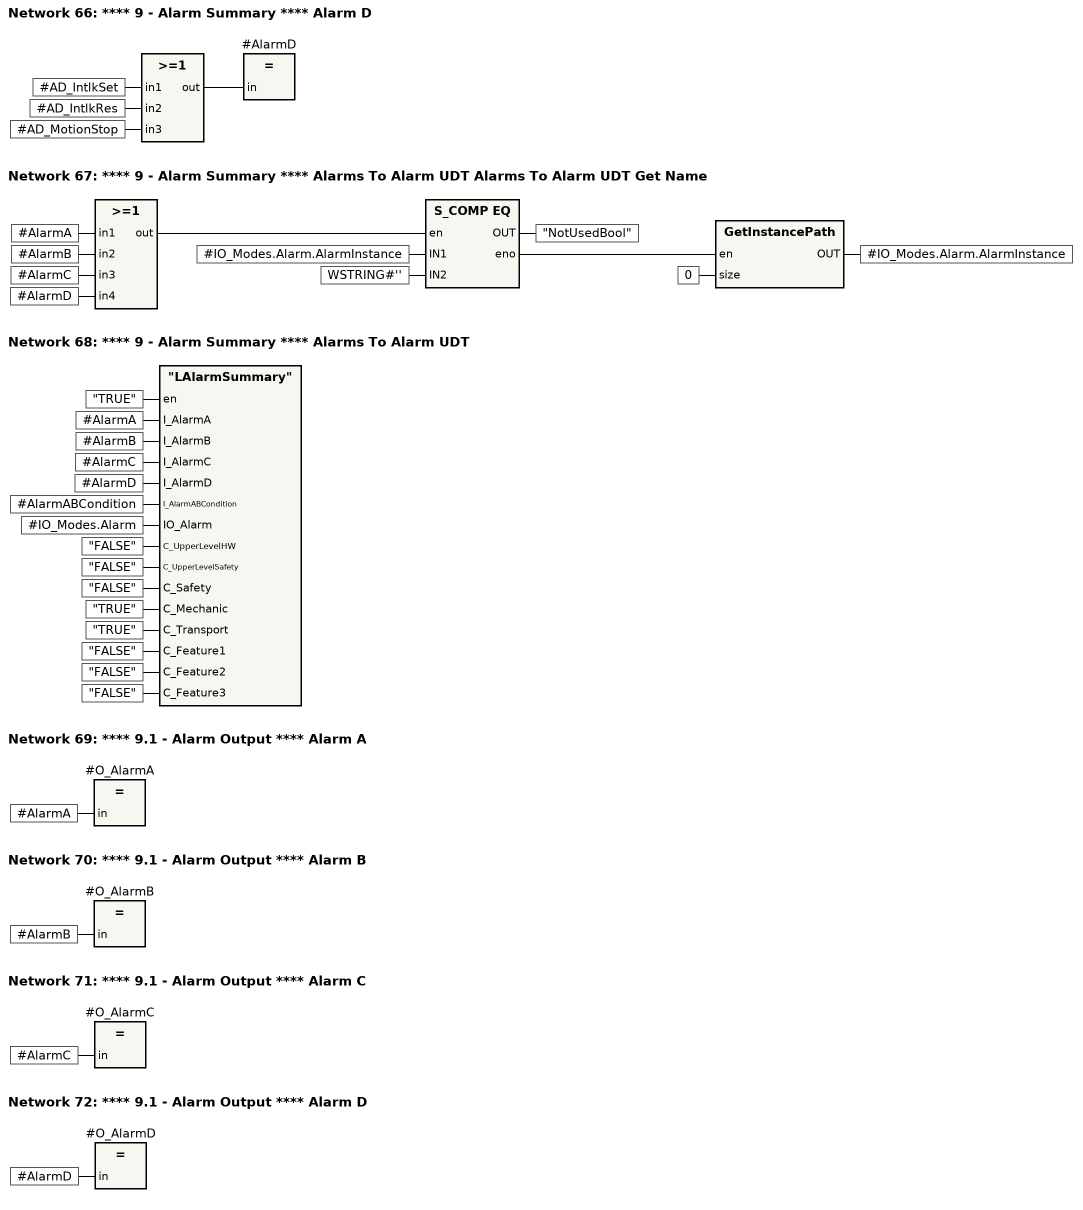
   #AlarmD := #AD_IntlkSet OR #AD_IntlkRes OR #AD_MotionStop;
END_REGION

REGION Network 67: **** 9 - Alarm Summary **** Alarms To Alarm UDT Alarms To Alarm UDT Get Name
   // Alarm D
   S_COMP(EN := #AlarmA OR #AlarmB OR #AlarmC OR #AlarmD,
          IN1 := #IO_Modes.Alarm.AlarmInstance,
          IN2 := WSTRING#'',
          OUT => "NotUsedBool",
          ENO => #_w1);
   IF #_w1 THEN GetInstancePath(size := 0, OUT => #IO_Modes.Alarm.AlarmInstance); END_IF;
END_REGION

REGION Network 68: **** 9 - Alarm Summary **** Alarms To Alarm UDT
   // Alarms To Alarm UDT
   IF "TRUE" THEN
       "LAlarmSummary"(I_AlarmA := #AlarmA,
                       I_AlarmB := #AlarmB,
                       I_AlarmC := #AlarmC,
                       I_AlarmD := #AlarmD,
                       I_AlarmABCondition := #AlarmABCondition,
                       IO_Alarm := #IO_Modes.Alarm,
                       C_UpperLevelHW := "FALSE",
                       C_UpperLevelSafety := "FALSE",
                       C_Safety := "FALSE",
                       C_Mechanic := "TRUE",
                       C_Transport := "TRUE",
                       C_Feature1 := "FALSE",
                       C_Feature2 := "FALSE",
                       C_Feature3 := "FALSE");
   END_IF;
END_REGION

REGION Network 69: **** 9.1 - Alarm Output **** Alarm A
   // Alarm A
   #O_AlarmA := #AlarmA;
END_REGION

REGION Network 70: **** 9.1 - Alarm Output **** Alarm B
   // Alarm B
   #O_AlarmB := #AlarmB;
END_REGION

REGION Network 71: **** 9.1 - Alarm Output **** Alarm C
   // Alarm C
   #O_AlarmC := #AlarmC;
END_REGION

REGION Network 72: **** 9.1 - Alarm Output **** Alarm D
   // Alarm D
   #O_AlarmD := #AlarmD;
END_REGION

REGION Network 73: **** 9.2 - Alarm DWord**** Alarm To DWord
   // Alarm To Word
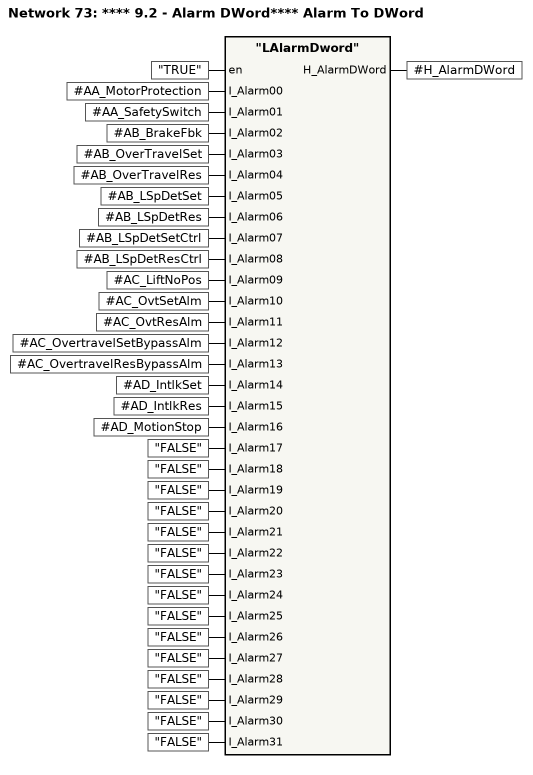
   IF "TRUE" THEN
       "LAlarmDword"(I_Alarm00 := #AA_MotorProtection,
                     I_Alarm01 := #AA_SafetySwitch,
                     I_Alarm02 := #AB_BrakeFbk,
                     I_Alarm03 := #AB_OverTravelSet,
                     I_Alarm04 := #AB_OverTravelRes,
                     I_Alarm05 := #AB_LSpDetSet,
                     I_Alarm06 := #AB_LSpDetRes,
                     I_Alarm07 := #AB_LSpDetSetCtrl,
                     I_Alarm08 := #AB_LSpDetResCtrl,
                     I_Alarm09 := #AC_LiftNoPos,
                     I_Alarm10 := #AC_OvtSetAlm,
                     I_Alarm11 := #AC_OvtResAlm,
                     I_Alarm12 := #AC_OvertravelSetBypassAlm,
                     I_Alarm13 := #AC_OvertravelResBypassAlm,
                     I_Alarm14 := #AD_IntlkSet,
                     I_Alarm15 := #AD_IntlkRes,
                     I_Alarm16 := #AD_MotionStop,
                     I_Alarm17 := "FALSE",
                     I_Alarm18 := "FALSE",
                     I_Alarm19 := "FALSE",
                     I_Alarm20 := "FALSE",
                     I_Alarm21 := "FALSE",
                     I_Alarm22 := "FALSE",
                     I_Alarm23 := "FALSE",
                     I_Alarm24 := "FALSE",
                     I_Alarm25 := "FALSE",
                     I_Alarm26 := "FALSE",
                     I_Alarm27 := "FALSE",
                     I_Alarm28 := "FALSE",
                     I_Alarm29 := "FALSE",
                     I_Alarm30 := "FALSE",
                     I_Alarm31 := "FALSE",
                     H_AlarmDWord => #H_AlarmDWord);
   END_IF;
END_REGION
END_FUNCTION_BLOCK
